ACTION MotorsActualPosition:
// Get Motors Actual Position
rMotorsActualPosition[1] := GVL_Motion.aMotors[1].GetPosition();
rMotorsActualPosition[2] := GVL_Motion.aMotors[2].GetPosition();
rMotorsActualPosition[3] := GVL_Motion.aMotors[3].GetPosition();
rValvesActualPosition[1] := GVL_Motion.aValvesObj[1].GetPosition();
rValvesActualPosition[2] := GVL_Motion.aValvesObj[2].GetPosition();
rValvesActualPosition[3] := GVL_Motion.aValvesObj[3].GetPosition();
rValvesActualPosition[4] := GVL_Motion.aValvesObj[4].GetPosition();
rValvesActualPosition[5] := GVL_Motion.aValvesObj[5].GetPosition();
rPumpsActualPosition[1] := GVL_Motion.aPumpsLinear[1].GetPosition();
rPumpsActualPosition[2] := GVL_Motion.aPumpsLinear[2].GetPosition();
rPumpsActualPosition[3] := GVL_Motion.aPumpsLinear[3].GetPosition();
rPumpsActualPosition[4] := GVL_Motion.aPumpsLinear[4].GetPosition();
rPumpsActualPosition[5] := GVL_Motion.aPumpsLinear[5].GetPosition();
rPumpsActualPosition[6] := GVL_Motion.aPumpsLinear[6].GetPosition();
rPumpsActualPosition[7] := GVL_Motion.aPumpsLinear[7].GetPosition();
rPumpsActualPosition[8] := GVL_Motion.aPumpsLinear[8].GetPosition();
rPumpsActualPosition[9] := GVL_Motion.aPumpsLinear[9].GetPosition();
rPumpsActualPosition[10] := GVL_Motion.aPumpsLinear[10].GetPosition();

//Linear Motors - M1, M2, M3
GVL_Motion.M1Motor.rActualPosition := F_ROUND_REAL(rInput := TO_REAL(rMotorsActualPosition[1]), iDecimalPlaces := 2)* -1;
GVL_Motion.M2Motor.rActualPosition := F_ROUND_REAL(rInput := TO_REAL(rMotorsActualPosition[2]), iDecimalPlaces := 2)* -1;
GVL_Motion.M3Motor.rActualPosition := F_ROUND_REAL(rInput := TO_REAL(rMotorsActualPosition[3]), iDecimalPlaces := 2)* -1;

//Vici Valves - M4 to M8
GVL_Motion.aValves[1].rActualPosition := F_ROUND_REAL(rInput := TO_REAL(rValvesActualPosition[1]), iDecimalPlaces := 2);
GVL_Motion.aValves[2].rActualPosition := F_ROUND_REAL(rInput := TO_REAL(rValvesActualPosition[2]), iDecimalPlaces := 2);
GVL_Motion.aValves[3].rActualPosition := F_ROUND_REAL(rInput := TO_REAL(rValvesActualPosition[3]), iDecimalPlaces := 2);
GVL_Motion.aValves[4].rActualPosition := F_ROUND_REAL(rInput := TO_REAL(rValvesActualPosition[4]), iDecimalPlaces := 2);
GVL_Motion.aValves[5].rActualPosition := F_ROUND_REAL(rInput := TO_REAL(rValvesActualPosition[5]), iDecimalPlaces := 2);

//Linear pumps - 1 to 10
GVL_Motion.aPumps[1].Linear.rActualPosition  := F_ROUND_REAL(rInput := TO_REAL(rPumpsActualPosition[1]), iDecimalPlaces := 2)* -1;
GVL_Motion.aPumps[2].Linear.rActualPosition  := F_ROUND_REAL(rInput := TO_REAL(rPumpsActualPosition[2]), iDecimalPlaces := 2)* -1;
GVL_Motion.aPumps[3].Linear.rActualPosition  := F_ROUND_REAL(rInput := TO_REAL(rPumpsActualPosition[3]), iDecimalPlaces := 2)* -1;
GVL_Motion.aPumps[4].Linear.rActualPosition  := F_ROUND_REAL(rInput := TO_REAL(rPumpsActualPosition[4]), iDecimalPlaces := 2)* -1;
GVL_Motion.aPumps[5].Linear.rActualPosition  := F_ROUND_REAL(rInput := TO_REAL(rPumpsActualPosition[5]), iDecimalPlaces := 2)* -1;
GVL_Motion.aPumps[6].Linear.rActualPosition  := F_ROUND_REAL(rInput := TO_REAL(rPumpsActualPosition[6]), iDecimalPlaces := 2)* -1;
GVL_Motion.aPumps[7].Linear.rActualPosition  := F_ROUND_REAL(rInput := TO_REAL(rPumpsActualPosition[7]), iDecimalPlaces := 2)* -1;
GVL_Motion.aPumps[8].Linear.rActualPosition  := F_ROUND_REAL(rInput := TO_REAL(rPumpsActualPosition[8]), iDecimalPlaces := 2)* -1;
GVL_Motion.aPumps[9].Linear.rActualPosition  := F_ROUND_REAL(rInput := TO_REAL(rPumpsActualPosition[9]), iDecimalPlaces := 2)* -1;
GVL_Motion.aPumps[10].Linear.rActualPosition := F_ROUND_REAL(rInput := TO_REAL(rPumpsActualPosition[10]), iDecimalPlaces := 2)* -1;
END_ACTION

ACTION MotorsJog:
//Manual Motors Moviment

//Manual Moviment motor 1 - Stage Collection Vertical Axis
GVL_Motion.aMotors[1].Jog(bFwd := GVL_HMI.ManualMov.bMotorsJogFwd[1], bBwd := GVL_HMI.ManualMov.bMotorsJogBwd[1]);
//Manual Moviment motor 2 - Sample Recovery Vertical Axis
GVL_Motion.aMotors[2].Jog(bFwd := GVL_HMI.ManualMov.bMotorsJogFwd[2], bBwd := GVL_HMI.ManualMov.bMotorsJogBwd[2]);
//Manual Moviment motor 3 - Sample Recovery Horizontal Axis
GVL_Motion.aMotors[3].Jog(bFwd := GVL_HMI.ManualMov.bMotorsJogFwd[3], bBwd := GVL_HMI.ManualMov.bMotorsJogBwd[3]);

//Manual Moviment M4 - Valve 1 
GVL_Motion.aValvesObj[1].Jog(bFwd := GVL_HMI.ManualMov.bValvesJogFwd[1], bBwd := GVL_HMI.ManualMov.bValvesJogBwd[1]);
//Manual Moviment M5 - Valve 2 
GVL_Motion.aValvesObj[2].Jog(bFwd := GVL_HMI.ManualMov.bValvesJogFwd[2], bBwd := GVL_HMI.ManualMov.bValvesJogBwd[2]);
//Manual Moviment M6 - Valve 3
GVL_Motion.aValvesObj[3].Jog(bFwd := GVL_HMI.ManualMov.bValvesJogFwd[3], bBwd := GVL_HMI.ManualMov.bValvesJogBwd[3]);
//Manual Moviment M7 - Valve 4
GVL_Motion.aValvesObj[4].Jog(bFwd := GVL_HMI.ManualMov.bValvesJogFwd[4], bBwd := GVL_HMI.ManualMov.bValvesJogBwd[4]);
//Manual Moviment M8 - Valve 5
GVL_Motion.aValvesObj[5].Jog(bFwd := GVL_HMI.ManualMov.bValvesJogFwd[5], bBwd := GVL_HMI.ManualMov.bValvesJogBwd[5]);

//Manual Moviment Pump 1 - Linear
GVL_Motion.aPumpsLinear[1].Jog(bFwd := GVL_HMI.ManualMov.bPumpsLinearJogFwd[1], bBwd := GVL_HMI.ManualMov.bPumpsLinearJogBwd[1]);
//Manual Moviment Pump 2 - Linear
GVL_Motion.aPumpsLinear[2].Jog(bFwd := GVL_HMI.ManualMov.bPumpsLinearJogFwd[2], bBwd := GVL_HMI.ManualMov.bPumpsLinearJogBwd[2]);
//Manual Moviment Pump 3 - Linear
GVL_Motion.aPumpsLinear[3].Jog(bFwd := GVL_HMI.ManualMov.bPumpsLinearJogFwd[3], bBwd := GVL_HMI.ManualMov.bPumpsLinearJogBwd[3]);
//Manual Moviment Pump 4 - Linear
GVL_Motion.aPumpsLinear[4].Jog(bFwd := GVL_HMI.ManualMov.bPumpsLinearJogFwd[4], bBwd := GVL_HMI.ManualMov.bPumpsLinearJogBwd[4]);
//Manual Moviment Pump 5 - Linear
GVL_Motion.aPumpsLinear[5].Jog(bFwd := GVL_HMI.ManualMov.bPumpsLinearJogFwd[5], bBwd := GVL_HMI.ManualMov.bPumpsLinearJogBwd[5]);
//Manual Moviment Pump 6 - Linear
GVL_Motion.aPumpsLinear[6].Jog(bFwd := GVL_HMI.ManualMov.bPumpsLinearJogFwd[6], bBwd := GVL_HMI.ManualMov.bPumpsLinearJogBwd[6]);
//Manual Moviment Pump 7 - Linear
GVL_Motion.aPumpsLinear[7].Jog(bFwd := GVL_HMI.ManualMov.bPumpsLinearJogFwd[7], bBwd := GVL_HMI.ManualMov.bPumpsLinearJogBwd[7]);
//Manual Moviment Pump 8 - Linear
GVL_Motion.aPumpsLinear[8].Jog(bFwd := GVL_HMI.ManualMov.bPumpsLinearJogFwd[8], bBwd := GVL_HMI.ManualMov.bPumpsLinearJogBwd[8]);
//Manual Moviment Pump 9 - Linear
GVL_Motion.aPumpsLinear[9].Jog(bFwd := GVL_HMI.ManualMov.bPumpsLinearJogFwd[9], bBwd := GVL_HMI.ManualMov.bPumpsLinearJogBwd[9]);
//Manual Moviment Pump 10 - Linear
GVL_Motion.aPumpsLinear[10].Jog(bFwd := GVL_HMI.ManualMov.bPumpsLinearJogFwd[10], bBwd := GVL_HMI.ManualMov.bPumpsLinearJogBwd[10]);
END_ACTION

METHOD Reset : BOOL
VAR_INPUT
END_VAR
VAR
	i : INT;
END_VAR
// ============================================================================
// PRG_ManualControl.Reset()
// ---------------------------------------------------------------------------
// Clears all manual commands, internal latches and FB states so that
// no manual movement can "resume" automatically when re-entering Manual Mode.
//
// This is a LOGIC reset only:
//  - Does NOT stop axes
//  - Does NOT reset axes
//  - Does NOT enable/disable drives
//
// Intended to be called from SystemInit.
// ============================================================================

// Default return
Reset := FALSE;

// ---------------------------------------------------------------------------
// 1) Reset HMI Manual Motor Commands (M1..M3)
// ---------------------------------------------------------------------------
FOR i := 1 TO 3 DO
    GVL_HMI.aManualMotorsCmd[i].bRun      := FALSE;
    GVL_HMI.aManualMotorsCmd[i].bStop     := FALSE;
    GVL_HMI.aManualMotorsCmd[i].iPosition := 0;
END_FOR

// ---------------------------------------------------------------------------
// 2) Reset HMI Manual Valve Commands (V1..V5)
// ---------------------------------------------------------------------------
FOR i := 1 TO 5 DO
    GVL_HMI.aManualValvesCmd[i].bMove      := FALSE;
    GVL_HMI.aManualValvesCmd[i].bStop      := FALSE;
    GVL_HMI.aManualValvesCmd[i].iTargetPos := 0;
END_FOR

// ---------------------------------------------------------------------------
// 3) Reset HMI Manual Pump Commands (P1..P10)
// ---------------------------------------------------------------------------
FOR i := 1 TO 10 DO
    GVL_HMI.aManualPumpsCmd[i].bActive    := FALSE;
    GVL_HMI.aManualPumpsCmd[i].rSpeed     := 0.0;
    GVL_HMI.aManualPumpsCmd[i].rVolume    := 0.0;
    GVL_HMI.aManualPumpsCmd[i].iDistance  := 0;
END_FOR

GVL_HMI.bRunPumpsBySpeedBt    := FALSE;
GVL_HMI.bRunPumpsByVolumeBt   := FALSE;
GVL_HMI.bRunPumpsByDistanceBt := FALSE;
GVL_HMI.bStopPumpsBt          := FALSE;

// ---------------------------------------------------------------------------
// 4) Reset internal pump control flags and arrays
// ---------------------------------------------------------------------------
bRunPumpsBySpeed    := FALSE;
bRunPumpsByVolume   := FALSE;
bRunPumpsByDistance := FALSE;

FOR i := 1 TO 10 DO
    aPumpsActivated[i] := FALSE;
    aPumpsSpeed[i]     := 0.0;
    aPumpsVolume[i]    := 0.0;
    aPumpsDistance[i]  := 0;
END_FOR

// ---------------------------------------------------------------------------
// 5) Reset interlock and auxiliary variables
// ---------------------------------------------------------------------------
bAllowMoveM2 := TRUE;
iTargetPosM2 := 0;
iM3Position  := 0;
rActualPosM3 := 0.0;

// ---------------------------------------------------------------------------
// 6) Reset FBs with internal state
// ---------------------------------------------------------------------------
fbPumpsController.Reset();   // assumes your FB has a Reset() method

// ---------------------------------------------------------------------------
// 7) Finalize
// ---------------------------------------------------------------------------
Reset := TRUE;
END_METHOD

END_PROGRAM

// ---- POUs/Functions/F_ROUND_REAL.TcPOU
FUNCTION F_ROUND_REAL : LREAL
VAR_INPUT
	rInput : LREAL;
  	iDecimalPlaces : INT;
END_VAR
VAR
	rFactor : LREAL;
    rScaled : LREAL;
    rRounded : LREAL;
END_VAR

rFactor := EXPT(10.0, iDecimalPlaces);         // Ex: 100.0 for 2 digits
rScaled := rInput * rFactor;

IF rScaled >= 0.0 THEN
    rRounded := TRUNC(rScaled + 0.5);
ELSE
    rRounded := TRUNC(rScaled - 0.5);
END_IF

F_ROUND_REAL := rRounded / rFactor;

END_FUNCTION

// ---- POUs/1. MachineControl/PRG_StoppedState.TcPOU
PROGRAM PRG_StoppedState

VAR_OUTPUT
    bStopAllMotorsDone : BOOL := FALSE; // TRUE when ALL axes (motors, valves, rotary pumps,
                     					// linear pumps) have completely finished stopping.
	                      				// Used by PRG_MasterControl to release SystemInit.
END_VAR

VAR
    // ------------------------------------------------------------------------
    // 1) HMI / Visual Feedback
    // ------------------------------------------------------------------------
    fbBlinkStartButton : FB_Blink;  // Blink logic for the Start button indicator
    
    // ------------------------------------------------------------------------
    // 2) Master Stop Execution Control
    // ------------------------------------------------------------------------
    bStopAllMotorsRequest : BOOL := FALSE;  
    // One-shot latch:
    // FALSE → stop request not yet triggered
    // TRUE  → stop request already armed; stop routine executing

    // ------------------------------------------------------------------------
    // 3) Per-axis STOP flags
    //    These arrays are used by ACTION ACT_StopAllMotors.
    //    TRUE  → axis still must be stopped (Stop() still being executed)
    //    FALSE → axis already fully stopped
    // ------------------------------------------------------------------------
    bStopMotors        : ARRAY[1..3]  OF BOOL;   // Linear motors M1..M3
    bStopValves        : ARRAY[1..5]  OF BOOL;   // Valves V1..V5
    bStopLinearPumps   : ARRAY[1..10] OF BOOL;   // Linear pump axes
    bStopRotaryPumps   : ARRAY[1..10] OF BOOL;   // Rotary pump axes

    // ------------------------------------------------------------------------
    // 4) Axis Status Structures
    //    Captured during ACTION ACT_ResetErrorMotors.
    // ------------------------------------------------------------------------
    stMotorStatus       : ARRAY[1..3]  OF ST_AxisReadStatus;
    stValveStatus       : ARRAY[1..5]  OF ST_AxisReadStatus;
    stLinearPumpStatus  : ARRAY[1..10] OF ST_AxisReadStatus;
    stRotaryPumpStatus  : ARRAY[1..10] OF ST_AxisReadStatus;

    // ------------------------------------------------------------------------
    // 5) Reset request guards for each axis
    //    TRUE  → Reset already attempted
    //    FALSE → Reset() still allowed to be triggered once
    // ------------------------------------------------------------------------
    aResetMotors       : ARRAY[1..3]  OF BOOL;
    aResetValves       : ARRAY[1..5]  OF BOOL;
    aResetLinearPumps  : ARRAY[1..10] OF BOOL;
    aResetRotaryPumps  : ARRAY[1..10] OF BOOL;

    // ------------------------------------------------------------------------
    // 6) Stop Monitoring Flags (used inside the refactored ACT_StopAllMotors)
    // ------------------------------------------------------------------------
    iAxis                    : INT;   // Generic loop index
    bIsNotMoving             : BOOL;  // Temporary axis movement flag
    bAllMotorsStopped        : BOOL;  // Group completion flags
    bAllValvesStopped        : BOOL;
    bAllRotaryPumpsStopped   : BOOL;
    bAllLinearPumpsStopped   : BOOL;

    // ------------------------------------------------------------------------
    // 7) Global Reset / StateMachine Control Flags
    // ------------------------------------------------------------------------ 
    bAllMotorsStop    : BOOL := FALSE;  // TRUE when all axes reached iNotMoving
    bAutoCycleReset   : BOOL := FALSE;  // TRUE when PRG_StateMachine.Reset() finished
    bCalibrationReset : BOOL := FALSE;  // TRUE when PRG_Calibration.Reset() finished
    bAllResetsDone    : BOOL := FALSE;  // TRUE when everything above is completed
	
	bAStopLogicLatchesDone	: BOOL := FALSE; // TRUE when as latches and flags were set to false
	
	i : INT; 

END_VAR

// ============================================================================
// PRG_StoppedState
// ----------------------------------------------------------------------------
// This program is executed while the machine is in the "Stopped" state.
// Responsibilities:
//  - Make the Start button blink when it is safe to start again
//  - Stop all axes (motors, valves, pumps) in a controlled way
//  - Reset axis errors
//  - Reset the AutoCycle and Calibration state machines
//  - Inform MasterControl when everything is fully reset (bAllResetsDone)
// ============================================================================

// ---------------------------------------------------------------------------
// Start Button Blink
//  - Blink only when: Safety is OK, all axes are stopped, and all resets done
//  - Output: GVL_IO.gDigOutputs.bStartIndicator
// ---------------------------------------------------------------------------
IF GVL_Safety.bSafetyEnable AND bStopAllMotorsDone AND bAStopLogicLatchesDone (*AND bAllResetsDone AND bCalibrationReset*) THEN 
    fbBlinkStartButton( bEnable := TRUE, tPeriod := T#1S );
ELSE
    fbBlinkStartButton( bEnable := FALSE, tPeriod := T#1S );
END_IF

GVL_IO.gDigOutputs.bStartIndicator := fbBlinkStartButton.bBlink;

// ---------------------------------------------------------------------------
// Reset axis errors
//  - Only executed after ALL motors have been confirmed as stopped
//  - This avoids resetting drives while they are still trying to stop
// ---------------------------------------------------------------------------
(*IF bAllMotorsStop THEN
    ACT_ResetErrorMotors();
END_IF
*)

IF NOT bAStopLogicLatchesDone THEN ACT_ResetCommandFlags(); END_IF


// ---------------------------------------------------------------------------
// Stop all axes
//  - This action:
//      * Sets stop requests for every axis (one-shot)
//      * Calls Stop() for each axis while it is moving
//      * Monitors when all stop requests are cleared
//      * Sets bStopAllMotorsDone when everything is stopped
// ---------------------------------------------------------------------------
ACT_StopAllMotors();

IF bStopAllMotorsDone THEN
    bAllMotorsStop := TRUE;     // All axes are now in a "not moving" state
END_IF
(*
// ---------------------------------------------------------------------------
// Reset AutoCycle State Machine
//  - PRG_StateMachine.Reset() should internally clear its own flags and states
//  - This is called until it returns TRUE once
// ---------------------------------------------------------------------------
IF NOT bAutoCycleReset THEN
    bAutoCycleReset := PRG_AutoCycle.Reset();
END_IF

// ---------------------------------------------------------------------------
// Reset Calibration Program
//  - PRG_Calibration.Reset() behaves similarly to PRG_StateMachine.Reset()
// ---------------------------------------------------------------------------
IF NOT bCalibrationReset THEN
    bCalibrationReset := PRG_Calibration.Reset();
END_IF

// ---------------------------------------------------------------------------
// Global done flag
//  - Used by MasterControl to know when StoppedState finished its job
//  - Only TRUE when:
//      * All axes are stopped   (bStopAllMotorsDone)
//      * AutoCycle reset is ok  (bAutoCycleReset)
//      * Calibration reset is ok(bCalibrationReset)
// ---------------------------------------------------------------------------
bAllResetsDone := bStopAllMotorsDone AND bAutoCycleReset AND bCalibrationReset;
*)

(* Before Tidy up from 05/12 
//Start Button Blink ------------------------------------------------
IF GVL_Safety.bSafetyEnable AND bStopAllMotorsDone AND bAllResetsDone THEN 
	fbBlinkStartButton( bEnable := TRUE, tPeriod := T#1S );
ELSE
	fbBlinkStartButton( bEnable := FALSE, tPeriod := T#1S );
END_IF

GVL_IO.gDigOutputs.bStartIndicator := fbBlinkStartButton.bBlink;

//Action to check if is there any motors with erros and reset them  
IF bAllMotorsStop THEN
	ACT_ResetErrorMotors();
END_IF

//Action to stop all motors 
ACT_StopAllMotors();

IF bStopAllMotorsDone THEN
	bAllMotorsStop := TRUE;
END_IF

//State Machine Reset
IF NOT bAutoCycleReset THEN
	bAutoCycleReset := PRG_StateMachine.Reset();
END_IF

//Calibration PRG Reset
IF NOT bCalibrationReset THEN
	bCalibrationReset := PRG_Calibration.Reset();
END_IF

bAllResetsDone := bStopAllMotorsDone AND bAutoCycleReset AND bCalibrationReset; *)

ACTION ACT_ResetCommandFlags:
(*
    Action: ACT_ResetCommandFlags
    Purpose:
        Clear all HMI command flags and internal latched commands that might remain TRUE
        after an abnormal interruption (STOP/Abort), preventing unintended auto-start
        when re-entering a mode.

    Where to call:
        - PRG_StoppedState (first scan / when entering STOPPED)
        - PRG_SystemInit (first scan / at init start)

    Notes:
        - This action is safe to call repeatedly (idempotent).
        - Adjust array bounds if your project differs.
*)

// ============================================================
// 1) Calibration - HMI triggers (buttons / commands)
// ============================================================
GVL_HMI.bStartCalibrationBt        := FALSE;

GVL_HMI.bCalLeakTestButton         := FALSE;
GVL_HMI.bCalPressureUpSystemBt     := FALSE;
GVL_HMI.bCalHoldSysPressureBt      := FALSE;
GVL_HMI.bCalStopLeakTestBt         := FALSE;

GVL_HMI.bCalLinearPumpsEnableBt    := FALSE;
GVL_HMI.bCalLinearPumpsHomeBt      := FALSE;
GVL_HMI.bCalLinearPumpsMoveBt      := FALSE;
GVL_HMI.bCalLinearPumpsStopBt      := FALSE;
GVL_HMI.bCalLinearPumpsDirty       := FALSE;

GVL_HMI.bCalMoveValves             := FALSE;
GVL_HMI.bCalMoveM1Motor            := FALSE;

// Scale / CalBox popups / acknowledge flags
GVL_HMI.bScaleNeedsAtention        := FALSE;
GVL_HMI.bScaleFixed                := FALSE;
GVL_HMI.bCalBoxNeedsAttention      := FALSE;
GVL_HMI.bCalBoxFixed               := FALSE;


// ============================================================
// 2) Calibration - internal latches (must be cleared on STOP/Init)
// ============================================================
GVL_Calibration.bStartCalibration      := FALSE;
GVL_Calibration.bAbortCalibration      := FALSE;
GVL_Calibration.bStartCreationCalJson  := FALSE;


// ============================================================
// 3) Manual Mode - motors / valves / pumps command arrays
// ============================================================

// Manual motors (adjust bounds if needed)
FOR i := 1 TO 3 DO
    GVL_HMI.aManualMotorsCmd[i].bRun  := FALSE;
    GVL_HMI.aManualMotorsCmd[i].bStop := FALSE;
END_FOR

// Manual valves
FOR i := 1 TO 5 DO
    GVL_HMI.aManualValvesCmd[i].bMove := FALSE;
    GVL_HMI.aManualValvesCmd[i].bStop := FALSE;
END_FOR

// Global pump buttons
GVL_HMI.bRunPumpsBySpeedBt  := FALSE;
GVL_HMI.bRunPumpsByVolumeBt := FALSE;

// Per-pump commands
FOR i := 1 TO 10 DO
    GVL_HMI.aManualPumpsCmd[i].bRunBySpeed  := FALSE;
    GVL_HMI.aManualPumpsCmd[i].bRunByVolume := FALSE;
    GVL_HMI.aManualPumpsCmd[i].bStop        := FALSE;
    GVL_HMI.aManualPumpsCmd[i].bActive      := FALSE;
END_FOR


// ============================================================
// 4) AutoCycle - popup/start/hold commands
// ============================================================
GVL_HMI.bShowAutoCyclePopup     	:= FALSE;
GVL_HMI.bStartAutoCycleButton   	:= FALSE;
GVL_HMI.bSystemReady_ReqAutoCycle 	:= FALSE;

GVL_HMI.bAutoCycleHoldReq       	:= FALSE;
GVL_HMI.bAutoCycleHoldActive    	:= FALSE;
GVL_HMI.bAutoCycleHoldPopup     	:= FALSE;
GVL_HMI.bAutoCycleContinueCmd   	:= FALSE;
GVL_HMI.bAutoCycleCancelCmd     	:= FALSE;


// ============================================================
// 5) Finishing
// ============================================================
bAStopLogicLatchesDone := TRUE;
END_ACTION

ACTION ACT_ResetErrorMotors:
// ============================================================================
// ACT_ResetErrorMotors
// ----------------------------------------------------------------------------
// Purpose:
//  1) Read status from all axis wrappers (motors, valves, pumps)
//  2) For each axis that is in Error, call its Reset() method once
//     - The aReset* arrays guarantee we do not repeatedly call Reset()
//     - Reset() is expected to return TRUE when the reset command has been sent
// ============================================================================

// ---------------------------------------------------------------------------
// 1) Read status from all axis wrappers
// ---------------------------------------------------------------------------

// Linear motors (M1..M3)
FOR iAxis := 1 TO 3 DO
    stMotorStatus[iAxis] := GVL_Motion.aMotors[iAxis].ReadStatus();
END_FOR

// Valves servo motors (V1..V5)
FOR iAxis := 1 TO 5 DO
    stValveStatus[iAxis] := GVL_Motion.aValvesObj[iAxis].ReadStatus();
END_FOR

// Linear pump motors (1..10)
FOR iAxis := 1 TO 10 DO
    stLinearPumpStatus[iAxis] := GVL_Motion.aPumpsLinear[iAxis].ReadStatus();
END_FOR

// Rotary pump motors (1..10)
FOR iAxis := 1 TO 10 DO
    stRotaryPumpStatus[iAxis] := GVL_Motion.aPumpsRotary[iAxis].ReadStatus();
END_FOR

// ---------------------------------------------------------------------------
// 2) For each axis in Error = TRUE, call Reset() once
//    The flag arrays (aReset*) are used as "one-shot" guards per axis.
// ---------------------------------------------------------------------------

// Linear motors

IF stMotorStatus[1].Error OR GVL_Motion.M1Motor.bMotionCommandsLocked THEN
	IF NOT aResetMotors[1] THEN
		aResetMotors[1] := GVL_Motion.aMotors[1].Reset();
	END_IF
END_IF

IF stMotorStatus[2].Error OR GVL_Motion.M2Motor.bMotionCommandsLocked THEN
	IF NOT aResetMotors[2] THEN
		aResetMotors[2] := GVL_Motion.aMotors[2].Reset();
	END_IF
END_IF

IF stMotorStatus[3].Error OR GVL_Motion.M3Motor.bMotionCommandsLocked THEN
	IF NOT aResetMotors[3] THEN
		aResetMotors[3] := GVL_Motion.aMotors[3].Reset();
	END_IF
END_IF

// Valves servo motors
FOR iAxis := 1 TO 5 DO
    IF stValveStatus[iAxis].Error OR GVL_Motion.aValves[iAxis].bMotionCommandsLocked THEN
        IF NOT aResetValves[iAxis] THEN
            aResetValves[iAxis] := GVL_Motion.aValvesObj[iAxis].Reset();
        END_IF
    END_IF
END_FOR

// Linear pump motors
FOR iAxis := 1 TO 10 DO
    IF stLinearPumpStatus[iAxis].Error OR GVL_Motion.aPumps[iAxis].Linear.bMotionCommandsLocked THEN
        IF NOT aResetLinearPumps[iAxis] THEN
            aResetLinearPumps[iAxis] := GVL_Motion.aPumpsLinear[iAxis].Reset();
        END_IF
    END_IF
END_FOR

// Rotary pump motors
FOR iAxis := 1 TO 10 DO
    IF stRotaryPumpStatus[iAxis].Error OR GVL_Motion.aPumps[iAxis].Rotary.bMotionCommandsLocked THEN
        IF NOT aResetRotaryPumps[iAxis] THEN
            aResetRotaryPumps[iAxis] := GVL_Motion.aPumpsRotary[iAxis].Reset();
        END_IF
    END_IF
END_FOR


(* Before Tidy up from 05/12
//Getting status from all motors
//Linear Motors
FOR i := 1 TO 3 DO
	stMotorStatus[i] := GVL_Motion.aMotors[i].ReadStatus();
END_FOR
//Valves Servo Motors
FOR i := 1 TO 5 DO
	stValveStatus[i] := GVL_Motion.aValvesObj[i].ReadStatus();
END_FOR
//Linear Pumps Motors
FOR i := 1 TO 10 DO
	stLinearPumpStatus[i] := GVL_Motion.aPumpsLinear[i].ReadStatus();
END_FOR
//Rotary Pumps Motors
FOR i := 1 TO 10 DO
	stRotaryPumpStatus[i] := GVL_Motion.aPumpsRotary[i].ReadStatus();
END_FOR

//Reset the motors that are in error
//Linear Motors
FOR i := 1 TO 3 DO
	IF stMotorStatus[i].Error THEN
		IF NOT aResetMotors[i] THEN
			aResetMotors[i] := GVL_Motion.aMotors[i].Reset();
		END_IF
	END_IF
END_FOR
//Valves Servo Motors
FOR i := 1 TO 5 DO
	IF stValveStatus[i].Error THEN
		IF NOT aResetValves[i] THEN
			aResetValves[i] := GVL_Motion.aValvesObj[i].Reset();
		END_IF
	END_IF
END_FOR
//Linear Pumps Motors
FOR i := 1 TO 10 DO
	IF stLinearPumpStatus[i].Error THEN
		IF NOT aResetLinearPumps[i] THEN
			aResetLinearPumps[i] := GVL_Motion.aPumpsLinear[i].Reset();
		END_IF
	END_IF
END_FOR
//Rotary Pumps Motors
FOR i := 1 TO 10 DO
	IF stRotaryPumpStatus[i].Error THEN
		IF NOT aResetRotaryPumps[i] THEN
			aResetRotaryPumps[i] := GVL_Motion.aPumpsRotary[i].Reset();
		END_IF
	END_IF
END_FOR*)
END_ACTION

ACTION ACT_StopAllMotors:
// ============================================================================
// ACT_StopAllMotors (Refactored)
// ----------------------------------------------------------------------------
// Purpose:
//  - Trigger a controlled stop for all motion axes:
//      * Linear motors (M1..M3)
//      * Valves servo motors (V1..V5)
//      * Rotary pumps (1..10)
//      * Linear pumps (1..10)
//  - Stop logic:
//      1) On first call (bStopAllMotorsRequest = FALSE), set all stop flags = TRUE
//      2) For each axis that is still moving, call its Stop() method
//      3) When Stop() returns TRUE, clear the corresponding flag to FALSE
//      4) When all flags are FALSE, set bStopAllMotorsDone = TRUE
// ============================================================================


// ---------------------------------------------------------------------------
// 1) One-shot: arm stop request for all axes
//    This block runs only once per StoppedState sequence.
// ---------------------------------------------------------------------------
IF NOT bStopAllMotorsRequest THEN
    // Linear motors
    bStopMotors[1] := NOT GVL_Motion.M1Motor.iNotMoving;      // Stop request for each linear motor
	bStopMotors[2] := NOT GVL_Motion.M2Motor.iNotMoving; 
	bStopMotors[3] := NOT GVL_Motion.M3Motor.iNotMoving; 
	
    // Valves servo motors
    FOR iAxis := 1 TO 5 DO
        bStopValves[iAxis] := NOT GVL_Motion.aValves[iAxis].iNotMoving;      // Stop request for each valve axis
    END_FOR

    // Linear pumps
    FOR iAxis := 1 TO 10 DO
        bStopLinearPumps[iAxis] := NOT GVL_Motion.aPumps[iAxis].Linear.iNotMoving; // Stop request for each linear pump axis
    END_FOR

    // Rotary pumps
    FOR iAxis := 1 TO 10 DO
        bStopRotaryPumps[iAxis] := NOT GVL_Motion.aPumps[iAxis].Rotary.iNotMoving; // Stop request for each rotary pump axis
    END_FOR
    
    bStopAllMotorsRequest := TRUE;       // One-shot armed
    bStopAllMotorsDone    := FALSE;      // Not done yet
END_IF


// ---------------------------------------------------------------------------
// 2) Call Stop() for each axis while it is still moving
//    Strategy:
//      - If axis is moving (iNotMoving = FALSE), keep requesting Stop()
//      - When Stop() returns TRUE, we clear the stop flag to FALSE
//      - If axis is already not moving, force the flag to FALSE
// ---------------------------------------------------------------------------

// --- Linear motors Stop - M1 to M3 -----------------------------------------
IF bStopMotors[1] THEN
	IF NOT GVL_Motion.M1Motor.iNotMoving THEN
		bStopMotors[1] := NOT GVL_Motion.aMotors[1].Stop();
	ELSE
		bStopMotors[1] := FALSE;
	END_IF
END_IF

IF bStopMotors[2] THEN
	IF NOT GVL_Motion.M2Motor.iNotMoving THEN
		bStopMotors[2] := NOT GVL_Motion.aMotors[2].Stop();
	ELSE
		bStopMotors[2] := FALSE;
	END_IF
END_IF
	

IF bStopMotors[3] THEN
	IF NOT GVL_Motion.M3Motor.iNotMoving THEN
		bStopMotors[3] := NOT GVL_Motion.aMotors[3].Stop();
	ELSE
		bStopMotors[3] := FALSE;
	END_IF
END_IF
	
// --- Valves Servo Motors Stop - V1 to V5 -----------------------------------
FOR iAxis := 1 TO 5 DO
	IF bStopValves[iAxis] THEN
		IF NOT GVL_Motion.aValves[iAxis].iNotMoving THEN
			bStopValves[iAxis] := NOT GVL_Motion.aValvesObj[iAxis].Stop();
		ELSE
			bStopValves[iAxis] := FALSE;
		END_IF
	END_IF
END_FOR


// --- Rotary Pumps Stop - 1 to 10 -------------------------------------------
//  - aPumps[x].Rotary.iNotMoving: feedback "axis moving" for each rotary pump
//  - aPumpsRotary[x].Stop(): Stop method on the pump rotary axis wrapper
FOR iAxis := 1 TO 10 DO
	IF  bStopRotaryPumps[iAxis] THEN
		IF NOT GVL_Motion.aPumps[iAxis].Rotary.iNotMoving THEN
			bStopRotaryPumps[iAxis] := NOT GVL_Motion.aPumpsRotary[iAxis].Stop();
		ELSE
			bStopRotaryPumps[iAxis] := FALSE;
		END_IF
	END_IF
END_FOR


// --- Linear Pumps Stop - 1 to 10 -------------------------------------------
//  - aPumps[x].Linear.iNotMoving: feedback "axis moving" for each linear pump
//  - aPumpsLinear[x].Stop(): Stop method on the linear pump axis wrapper
FOR iAxis := 1 TO 10 DO
	IF bStopLinearPumps[iAxis] THEN
		IF NOT GVL_Motion.aPumps[iAxis].Linear.iNotMoving THEN
			bStopLinearPumps[iAxis] := NOT GVL_Motion.aPumpsLinear[iAxis].Stop();
		ELSE
			bStopLinearPumps[iAxis] := FALSE;
		END_IF
	END_IF
END_FOR


// ---------------------------------------------------------------------------
// 3) Global "done" condition for stopping all axes
//    When no stop flag is active in any group, all axes are considered stopped.
// ---------------------------------------------------------------------------

// Check linear motors

bAllMotorsStopped := NOT bStopMotors[1] AND NOT bStopMotors[2] AND NOT bStopMotors[3];


// Check valves
bAllValvesStopped := TRUE;
FOR iAxis := 1 TO 5 DO
    bAllValvesStopped := bAllValvesStopped AND NOT bStopValves[iAxis];
END_FOR

// Check rotary pumps
bAllRotaryPumpsStopped := TRUE;
FOR iAxis := 1 TO 10 DO
    bAllRotaryPumpsStopped := bAllRotaryPumpsStopped AND NOT bStopRotaryPumps[iAxis];
END_FOR

// Check linear pumps
bAllLinearPumpsStopped := TRUE;
FOR iAxis := 1 TO 10 DO
    bAllLinearPumpsStopped := bAllLinearPumpsStopped AND NOT bStopLinearPumps[iAxis];
END_FOR

// Final global flag
bStopAllMotorsDone := bAllMotorsStopped
                      AND bAllValvesStopped
                      AND bAllRotaryPumpsStopped
                      AND bAllLinearPumpsStopped;


(* Before Tidy up from 05/12
//Stop all motors. Linear, valves, pumps.
IF NOT bStopAllMotorsRequest THEN
	FOR i := 1 TO 3 DO
		bStopMotors[i] := TRUE; //Stop Request for every motor turn true
	END_FOR
	FOR i := 1 TO 5 DO
		bStopValves[i] := TRUE;
	END_FOR
	FOR i := 1 TO 10 DO
		bStopLinearPumps[i] := TRUE;
	END_FOR
	FOR i := 1 TO 10 DO
		bStopRotaryPumps[i] := TRUE;
	END_FOR
	
	bStopAllMotorsRequest	:= TRUE;
	bStopAllMotorsDone		:= FALSE;
END_IF

//Every Motor Method Stop() call
//Linear Motors Stop - M1 to M3
IF NOT GVL_Motion.M1Motor.iNotMoving THEN
	bStopMotors[1] := NOT GVL_Motion.aMotors[1].Stop();
ELSE
	bStopMotors[1] := FALSE;
END_IF

IF NOT GVL_Motion.M2Motor.iNotMoving THEN
	bStopMotors[2] := NOT GVL_Motion.aMotors[2].Stop();
ELSE
	bStopMotors[2] := FALSE;
END_IF


IF NOT GVL_Motion.M3Motor.iNotMoving THEN
	bStopMotors[3] := NOT GVL_Motion.aMotors[3].Stop();
ELSE
	bStopMotors[3] := FALSE;
END_IF

//Valve Servo Motors Stop - M4 to M8
IF NOT GVL_Motion.aValves[1].iNotMoving THEN
	bStopValves[1] := NOT GVL_Motion.aValvesObj[1].Stop();
ELSE
	bStopValves[1] := FALSE;
END_IF

IF NOT GVL_Motion.aValves[2].iNotMoving THEN
	bStopValves[2] := NOT GVL_Motion.aValvesObj[2].Stop();
ELSE
	bStopValves[2] := FALSE;
END_IF

IF NOT GVL_Motion.aValves[3].iNotMoving THEN
	bStopValves[3] := NOT GVL_Motion.aValvesObj[3].Stop();
ELSE
	bStopValves[3] := FALSE;
END_IF

IF NOT GVL_Motion.aValves[4].iNotMoving THEN
	bStopValves[4] := NOT GVL_Motion.aValvesObj[4].Stop();
ELSE
	bStopValves[4] := FALSE;
END_IF

IF NOT GVL_Motion.aValves[5].iNotMoving THEN
	bStopValves[5] := NOT GVL_Motion.aValvesObj[5].Stop();
ELSE
	bStopValves[5] := FALSE;
END_IF

//Rotary Pumps Stop - 1 to 10
IF NOT GVL_Motion.aPumps[1].Rotary.iNotMoving THEN
	bStopRotaryPumps[1] := NOT GVL_Motion.aPumpsRotary[1].Stop();
ELSE
	bStopRotaryPumps[1] := FALSE;
END_IF

IF NOT GVL_Motion.aPumps[2].Rotary.iNotMoving THEN
	bStopRotaryPumps[2] := NOT GVL_Motion.aPumpsRotary[2].Stop();
ELSE
	bStopRotaryPumps[2] := FALSE;
END_IF

IF NOT GVL_Motion.aPumps[3].Rotary.iNotMoving THEN
	bStopRotaryPumps[3] := NOT GVL_Motion.aPumpsRotary[3].Stop();
ELSE
	bStopRotaryPumps[3] := FALSE;
END_IF

IF NOT GVL_Motion.aPumps[4].Rotary.iNotMoving THEN
	bStopRotaryPumps[4] := NOT GVL_Motion.aPumpsRotary[4].Stop();
ELSE
	bStopRotaryPumps[4] := FALSE;
END_IF

IF NOT GVL_Motion.aPumps[5].Rotary.iNotMoving THEN
	bStopRotaryPumps[5] := NOT GVL_Motion.aPumpsRotary[5].Stop();
ELSE
	bStopRotaryPumps[5] := FALSE;
END_IF

IF NOT GVL_Motion.aPumps[6].Rotary.iNotMoving THEN
	bStopRotaryPumps[6] := NOT GVL_Motion.aPumpsRotary[6].Stop();
ELSE
	bStopRotaryPumps[6] := FALSE;
END_IF

IF NOT GVL_Motion.aPumps[7].Rotary.iNotMoving THEN
	bStopRotaryPumps[7] := NOT GVL_Motion.aPumpsRotary[7].Stop();
ELSE
	bStopRotaryPumps[7] := FALSE;
END_IF

IF NOT GVL_Motion.aPumps[8].Rotary.iNotMoving THEN
	bStopRotaryPumps[8] := NOT GVL_Motion.aPumpsRotary[8].Stop();
ELSE
	bStopRotaryPumps[8] := FALSE;
END_IF

IF NOT GVL_Motion.aPumps[9].Rotary.iNotMoving THEN
	bStopRotaryPumps[9] := NOT GVL_Motion.aPumpsRotary[9].Stop();
ELSE
	bStopRotaryPumps[9] := FALSE;
END_IF

IF NOT GVL_Motion.aPumps[10].Rotary.iNotMoving THEN
	bStopRotaryPumps[10] := NOT GVL_Motion.aPumpsRotary[10].Stop();
ELSE
	bStopRotaryPumps[10] := FALSE;
END_IF

//Linear Pumps Stop - 1 to 10
IF NOT GVL_Motion.aPumps[1].Linear.iNotMoving THEN
	bStopLinearPumps[1] := NOT GVL_Motion.aPumpsLinear[1].Stop();
ELSE
	bStopLinearPumps[1] := FALSE;
END_IF

IF NOT GVL_Motion.aPumps[2].Linear.iNotMoving THEN
	bStopLinearPumps[2] := NOT GVL_Motion.aPumpsLinear[2].Stop();
ELSE
	bStopLinearPumps[2] := FALSE;
END_IF

IF NOT GVL_Motion.aPumps[3].Linear.iNotMoving THEN
	bStopLinearPumps[3] := NOT GVL_Motion.aPumpsLinear[3].Stop();
ELSE
	bStopLinearPumps[3] := FALSE;
END_IF

IF NOT GVL_Motion.aPumps[4].Linear.iNotMoving THEN
	bStopLinearPumps[4] := NOT GVL_Motion.aPumpsLinear[4].Stop();
ELSE
	bStopLinearPumps[4] := FALSE;
END_IF

IF NOT GVL_Motion.aPumps[5].Linear.iNotMoving THEN
	bStopLinearPumps[5] := NOT GVL_Motion.aPumpsLinear[5].Stop();
ELSE
	bStopLinearPumps[5] := FALSE;
END_IF

IF NOT GVL_Motion.aPumps[6].Linear.iNotMoving THEN
	bStopLinearPumps[6] := NOT GVL_Motion.aPumpsLinear[6].Stop();
ELSE
	bStopLinearPumps[6] := FALSE;
END_IF

IF NOT GVL_Motion.aPumps[7].Linear.iNotMoving THEN
	bStopLinearPumps[7] := NOT GVL_Motion.aPumpsLinear[7].Stop();
ELSE
	bStopLinearPumps[7] := FALSE;
END_IF

IF NOT GVL_Motion.aPumps[8].Linear.iNotMoving THEN
	bStopLinearPumps[8] := NOT GVL_Motion.aPumpsLinear[8].Stop();
ELSE
	bStopLinearPumps[8] := FALSE;
END_IF

IF NOT GVL_Motion.aPumps[9].Linear.iNotMoving THEN
	bStopLinearPumps[9] := NOT GVL_Motion.aPumpsLinear[9].Stop();
ELSE
	bStopLinearPumps[9] := FALSE;
END_IF

IF NOT GVL_Motion.aPumps[10].Linear.iNotMoving THEN
	bStopLinearPumps[10] := NOT GVL_Motion.aPumpsLinear[10].Stop();
ELSE
	bStopLinearPumps[10] := FALSE;
END_IF

IF NOT bStopMotors[1] AND NOT bStopMotors[2] AND NOT bStopMotors[3] THEN
	IF NOT bStopValves[1] AND NOT bStopValves[2] AND NOT bStopValves[3] AND NOT bStopValves[4] AND NOT bStopValves[5] THEN
		IF NOT bStopRotaryPumps[1] AND NOT bStopRotaryPumps[2] AND NOT bStopRotaryPumps[3] AND NOT bStopRotaryPumps[4] AND NOT bStopRotaryPumps[5] AND NOT bStopRotaryPumps[6] AND NOT bStopRotaryPumps[7] AND NOT bStopRotaryPumps[8] AND NOT bStopRotaryPumps[9] AND NOT bStopRotaryPumps[10] THEN
			IF NOT bStopLinearPumps[1] AND NOT bStopLinearPumps[2] AND NOT bStopLinearPumps[3] AND NOT bStopLinearPumps[4] AND NOT bStopLinearPumps[5] AND NOT bStopLinearPumps[6] AND NOT bStopLinearPumps[7] AND NOT bStopLinearPumps[8] AND NOT bStopLinearPumps[9] AND NOT bStopLinearPumps[10] THEN
				bStopAllMotorsDone		:= TRUE;
			END_IF
		END_IF
	END_IF
END_IF
*)
END_ACTION

METHOD Reset : BOOL
VAR_INPUT
END_VAR
// ============================================================================
// Reset()
// ----------------------------------------------------------------------------
// Purpose:
//  - Clear all internal flags and arrays of PRG_StoppedState
//  - Prepare this program to run a new full stopped-sequence
// Behavior:
//  - Sets all internal booleans and arrays to FALSE
//  - Returns TRUE once, when the reset conditions are satisfied
//    (here: simply when there is no stop request and no "done" flag)
// ============================================================================

// ---------------------------------------------------------------------------
// 1) Reset main flags
// ---------------------------------------------------------------------------
bStopAllMotorsRequest := FALSE;
bStopAllMotorsDone    := FALSE;

bAllMotorsStop          := FALSE;
bAutoCycleReset         := FALSE;
bCalibrationReset       := FALSE;
bAllResetsDone          := FALSE;
bAStopLogicLatchesDone  := FALSE;

// ---------------------------------------------------------------------------
// 2) Reset arrays used in error reset / stop logic
// ---------------------------------------------------------------------------
// Motors reset flags
FOR iAxis := 1 TO 3 DO
    aResetMotors[iAxis] := FALSE;
END_FOR

// Valves reset flags
FOR iAxis := 1 TO 5 DO
    aResetValves[iAxis] := FALSE;
END_FOR

// Linear pumps reset flags
FOR iAxis := 1 TO 10 DO
    aResetLinearPumps[iAxis] := FALSE;
END_FOR

// Rotary pumps reset flags
FOR iAxis := 1 TO 10 DO
    aResetRotaryPumps[iAxis] := FALSE;
END_FOR

// ---------------------------------------------------------------------------
// 3) Return value
//    - With the current logic, right after executing this method
//      both bStopAllMotorsRequest and bStopAllMotorsDone are FALSE
//      so Reset = TRUE will be returned.
// ---------------------------------------------------------------------------
IF NOT bStopAllMotorsRequest AND NOT bStopAllMotorsDone THEN
    Reset := TRUE;
    RETURN;
ELSE
    Reset := FALSE;
END_IF
END_METHOD

END_PROGRAM

// ---- POUs/1. MachineControl/PRG_SystemReady.TcPOU
PROGRAM PRG_SystemReady
VAR_OUTPUT
	bSystemReadyToStart : BOOL;      // TRUE when machine is ready to accept Start 	 	
END_VAR
VAR
	fbBlinkStartButton      : FB_Blink;
    fbBlinkMachineModeName  : FB_Blink;

    bRecipeCorrectLoaded    : BOOL := FALSE;
    bSettingsCorrectLoaded  : BOOL := FALSE;

    rTrigStartButton        : R_TRIG;    // Rising edge for main Start button
    rTrigPopupStartBtn      : R_TRIG;    // Rising edge for popup "Start Auto Cycle" button
	
END_VAR

// ============================================================================
// 0) Default: no request to Auto Cycle unless logic sets it here
// ============================================================================
GVL_HMI.bSystemReady_ReqAutoCycle := FALSE;

// ============================================================================
// 1) Basic "System Ready" condition & Start button blinking
//    - Only blink Start when safety is OK, no incoherence and data loaded
// ============================================================================

// Conditions for "ready to start" as you prefer
IF GVL_Safety.bSafetyEnable
   AND NOT GVL_HMI.bIncoherenceDetected THEN
    bSystemReadyToStart := TRUE;
ELSE
    bSystemReadyToStart := FALSE;
END_IF

// Start button blinking only when system is ready
fbBlinkStartButton(
    bEnable := bSystemReadyToStart,
    tPeriod := T#1S
);
GVL_IO.gDigOutputs.bStartIndicator := fbBlinkStartButton.bBlink;

// ============================================================================
// 2) Handle main Start button on System Ready
//    - Rising edge on Start button
//    - If "ready to start" -> open popup for comment
//    - If not ready / incoherence -> raise alert (same behavior as before)
// ============================================================================

rTrigStartButton(CLK := GVL_IO.gDigInputs.bStartButton);

IF rTrigStartButton.Q THEN
    IF bSystemReadyToStart THEN
        // No incoherence and everything loaded: request popup for comment
        GVL_HMI.bShowAutoCyclePopup   := TRUE;
        GVL_HMI.bIncoherenceAlert     := FALSE;

        // Optionally clear previous comment and reset popup button
        GVL_HMI.sAutoCycleComment     := '';
        GVL_HMI.bStartAutoCycleButton := FALSE;
    ELSE
        // Not ready: keep the "old behavior": show incoherence / warning
        GVL_HMI.bIncoherenceAlert := TRUE;
    END_IF
END_IF

// ============================================================================
// 3) Handle popup "Start Auto Cycle" button
//    - Rising edge on bStartAutoCycleButton
//    - Double-check safety, incoherence and comment length
//    - If OK -> raise bSystemReady_ReqAutoCycle (one-shot)
// ============================================================================

rTrigPopupStartBtn(CLK := GVL_HMI.bStartAutoCycleButton);

IF rTrigPopupStartBtn.Q THEN

    // Extra safety: conditions may have changed since popup was opened
    IF GVL_Safety.bSafetyEnable
       AND NOT GVL_HMI.bIncoherenceDetected
       AND (LEN(GVL_HMI.sAutoCycleComment) > 0) THEN

        // All good: request transition to AUTO_CYCLE
        GVL_HMI.bSystemReady_ReqAutoCycle := TRUE;

        // Close popup
        GVL_HMI.bShowAutoCyclePopup := FALSE;

        // Optionally keep comment for logging

    ELSE
        // Something is wrong:
        // - Safety disabled
        // - Incoherence detected
        // - Or empty comment
        IF GVL_HMI.bIncoherenceDetected THEN
            GVL_HMI.bIncoherenceAlert := TRUE;
        END_IF

        // Reset popup start button, keep popup open so the user can fix it
        GVL_HMI.bStartAutoCycleButton := FALSE;
    END_IF

END_IF

END_PROGRAM

// ---- POUs/Utilities/PRG_UpdateVariablesMoving.TcPOU
PROGRAM PRG_UpdateVariablesMoving
VAR
	bFirstVariablesAssignment  : BOOL := FALSE;
	bValvesSettingsAssignment  : BOOL := FALSE;
	bPumpsFactorAssignment	   : BOOL := FALSE;
	bPumpsSettingsAssignment   : BOOL := FALSE;
	bPumpsDeadVolumeAssignment : BOOL := FALSE;
	
	i : UINT := 1;
	
	aDebug	: ARRAY[1..10] OF BOOL;
	bUpdatePumpFactor	: BOOL := FALSE;
	
END_VAR

IF NOT GVL_IO.gDigInputs.bAccessDoor4InterlockFdbk AND NOT GVL_IO.gDigInputs.bAccessDoor5InterlockFdbk AND NOT GVL_IO.gDigInputs.bAccessDoor6InterlockFdbk THEN
	GVL_Safety.SafetyOutputs.bBelowDoorsFeedback := TRUE;
ELSE
	GVL_Safety.SafetyOutputs.bBelowDoorsFeedback := FALSE;
END_IF

// Mapping bellow doors signals as they are not in safety DI
(*
GVL_IO.gRelayOutputs.bSampleRecoveryLight 		:= NOT GVL_Safety.bTopDoorsClosedFeedback;
GVL_IO.gRelayOutputs.bStageCollectionLeftLight 	:= NOT GVL_Safety.bTopDoorsClosedFeedback;
GVL_IO.gRelayOutputs.bStageCollectionRightLight := NOT GVL_Safety.bTopDoorsClosedFeedback;
*)

// Vial Rack position check
IF GVL_IO.gProfinetInput.iCurrentValue > 120000 THEN
	GVL_IO.bVialRackPresent := TRUE;
ELSE
	GVL_IO.bVialRackPresent := FALSE;
END_IF

// Valves Settings Assignment
IF NOT bValvesSettingsAssignment THEN
	FOR i := 1 TO 5 DO
		GVL_Motion.aValves[i].rTargetVel := 600;
		GVL_Motion.aValves[i].rAcceleration := 200;
		GVL_Motion.aValves[i].rDeceleration := 200;
	END_FOR
	bValvesSettingsAssignment := TRUE;
END_IF

//Pumps factor Assignment [ml/rev]
IF NOT bPumpsFactorAssignment OR bUpdatePumpFactor THEN

	FOR i := 1 TO 10 DO
		GVL_Motion.aPumps[i].Rotary.rPumpFactorFillJars 	:= GVL_Retain.aCalibrationPumpFactor[i];
		GVL_Motion.aPumps[i].Rotary.rPumpFactorFillCalBox 	:= GVL_Retain.aCalibrationPumpFactor[i];
		GVL_Motion.aPumps[i].Rotary.rPumpFactorFromCalBox	:= GVL_Retain.aCalibrationPumpFactor[i];
	END_FOR
		
	bPumpsFactorAssignment := TRUE;
END_IF

//Pumps line dead Volume pipes/tubing Assignment [ml]
IF NOT bPumpsDeadVolumeAssignment THEN
	GVL_Motion.aPumps[1].Rotary.rDeadVolume := -0.3;//4.5;//10.0;
	GVL_Motion.aPumps[2].Rotary.rDeadVolume := -0.5;//8.0;//10.0;
	GVL_Motion.aPumps[3].Rotary.rDeadVolume := 0.65;//5.5;//27.0;
	GVL_Motion.aPumps[4].Rotary.rDeadVolume := 0.2;//6.5;//19.0;
	GVL_Motion.aPumps[5].Rotary.rDeadVolume := 2.3;//10.5;//14.0;
	GVL_Motion.aPumps[6].Rotary.rDeadVolume := 0.65;//7.5;//21.0;
	GVL_Motion.aPumps[7].Rotary.rDeadVolume := 0.85;//8.3;//21.0;
	GVL_Motion.aPumps[8].Rotary.rDeadVolume := -0.3;//6.0;//12.0;
	GVL_Motion.aPumps[9].Rotary.rDeadVolume := 1.4;//7.9;//16.0;
	GVL_Motion.aPumps[10].Rotary.rDeadVolume := 0.8;//8.1;//16.0;
END_IF

//Pumps Settings Assignment
IF NOT bPumpsSettingsAssignment THEN
	FOR i := 1 TO 10 DO
		GVL_Motion.aPumps[i].Rotary.rSpeed := 1800; //1800º/sec with is equal to 300 revs/min
		GVL_Motion.aPumps[i].Rotary.rAcceleration := 2000; //Standard Acceleration based on motor speed
		GVL_Motion.aPumps[i].Rotary.rDeceleration := 2000; //Standard Acceleration based on motor speed
	END_FOR
	bPumpsSettingsAssignment := TRUE;
END_IF

//Pumps Home sensor bit
GVL_Motion.aPumps[1].Linear.bHomeSensorState := GVL_Motion.aPumps[1].Linear.iHomeSensor.0; 
GVL_Motion.aPumps[2].Linear.bHomeSensorState := GVL_Motion.aPumps[2].Linear.iHomeSensor.0; 
GVL_Motion.aPumps[3].Linear.bHomeSensorState := GVL_Motion.aPumps[3].Linear.iHomeSensor.0; 
GVL_Motion.aPumps[4].Linear.bHomeSensorState := GVL_Motion.aPumps[4].Linear.iHomeSensor.0; 
GVL_Motion.aPumps[5].Linear.bHomeSensorState := GVL_Motion.aPumps[5].Linear.iHomeSensor.0; 
GVL_Motion.aPumps[6].Linear.bHomeSensorState := GVL_Motion.aPumps[6].Linear.iHomeSensor.0; 
GVL_Motion.aPumps[7].Linear.bHomeSensorState := GVL_Motion.aPumps[7].Linear.iHomeSensor.0; 
GVL_Motion.aPumps[8].Linear.bHomeSensorState := GVL_Motion.aPumps[8].Linear.iHomeSensor.0; 
GVL_Motion.aPumps[9].Linear.bHomeSensorState := GVL_Motion.aPumps[9].Linear.iHomeSensor.0; 
GVL_Motion.aPumps[10].Linear.bHomeSensorState := GVL_Motion.aPumps[10].Linear.iHomeSensor.0; 

// Pump factor Restore
IF aDebug[1] THEN
	GVL_Retain.aCalibrationPumpFactor[1] := 0.1;
END_IF
IF aDebug[2] THEN
	GVL_Retain.aCalibrationPumpFactor[2] := 0.1;
END_IF
IF aDebug[3] THEN
	GVL_Retain.aCalibrationPumpFactor[3] := 0.1;
END_IF
IF aDebug[4] THEN
	GVL_Retain.aCalibrationPumpFactor[4] := 0.1;
END_IF
IF aDebug[5] THEN
	GVL_Retain.aCalibrationPumpFactor[5] := 0.1;
END_IF
IF aDebug[6] THEN
	GVL_Retain.aCalibrationPumpFactor[6] := 0.1;
END_IF
IF aDebug[7] THEN
	GVL_Retain.aCalibrationPumpFactor[7] := 0.1;
END_IF
IF aDebug[8] THEN
	GVL_Retain.aCalibrationPumpFactor[8] := 0.1;
END_IF
IF aDebug[9] THEN
	GVL_Retain.aCalibrationPumpFactor[9] := 0.1;
END_IF
IF aDebug[10] THEN
	GVL_Retain.aCalibrationPumpFactor[10] := 0.1;
END_IF


// temporary until we are able to get this parameter from hmi or configuration File **************************************************************************
IF NOT bFirstVariablesAssignment THEN
	//Default Homing Motors settings
	GVL_Motion.M1Motor.rHomeAcc 	:= 20.0;
	GVL_Motion.M1Motor.rHomeDec 	:= 20.0;
	GVL_Motion.M1Motor.rHomeVel 	:= 15.0;
	GVL_Motion.M2Motor.rHomeAcc 	:= 20.0;
	GVL_Motion.M2Motor.rHomeDec 	:= 20.0;
	GVL_Motion.M2Motor.rHomeVel 	:= 15.0;
	GVL_Motion.M3Motor.rHomeAcc 	:= 20.0;
	GVL_Motion.M3Motor.rHomeDec 	:= 20.0;
	GVL_Motion.M3Motor.rHomeVel 	:= 15.0;
	
	FOR i :=1 TO 5 DO
		GVL_Motion.aValves[i].rHomeAcc := 400.0;
		GVL_Motion.aValves[i].rHomeDec := 400.0;
		GVL_Motion.aValves[i].rHomeVel := 500.0;
	END_FOR
	
	FOR i :=1 TO 10 DO
		GVL_Motion.aPumps[i].Linear.rHomeAcc := 100.0;
		GVL_Motion.aPumps[i].Linear.rHomeDec := 100.0;
		GVL_Motion.aPumps[i].Linear.rHomeVel := 200.0;
	END_FOR
	
	GVL_Settings.stMachineParam.fM1PositionDeceleration := 30;
	
	bFirstVariablesAssignment := TRUE;
	(*
	GVL_Retain.rLinearPumpOldPosition[1] := -700.0;
	GVL_Retain.rLinearPumpOldPosition[2] := -700.0;
	GVL_Retain.rLinearPumpOldPosition[3] := -700.0;
	GVL_Retain.rLinearPumpOldPosition[4] := -700.0;
	GVL_Retain.rLinearPumpOldPosition[5] := -700.0;
	GVL_Retain.rLinearPumpOldPosition[6] := -700.0;
	GVL_Retain.rLinearPumpOldPosition[7] := -700.0;
	GVL_Retain.rLinearPumpOldPosition[8] := -700.0;
	GVL_Retain.rLinearPumpOldPosition[9] := -700.0;
	GVL_Retain.rLinearPumpOldPosition[10] := -700.0;
	*)
	
END_IF

END_PROGRAM

// ---- POUs/1. MachineControl/PRG_SafetyHandle.TcPOU
PROGRAM PRG_SafetyHandle
VAR
	//Air Supply testing
	bAirSupplyEnable: BOOL	:= TRUE;
	bAirSupplyReset	: BOOL	:= FALSE;
	
	bLockDoors	  	: BOOL 	:= FALSE;	   	// Variable that sends the lock doors signal
	
	tonStabilizingFaults : TON;
	tonClearFaults		 : TON;
	
	i	: USINT;
END_VAR

//Safety Restart & Error Ack
IF GVL_Safety.SafetyInputs.bMachineReset OR GVL_Safety.bM1STOErrorAck THEN
	GVL_Safety.bSafetyErrorAck			:= TRUE;
	GVL_Motion.M1Motor.bTS_ErrorAck		:= TRUE;
ELSE
	GVL_Safety.bSafetyErrorAck			:= FALSE;
	GVL_Motion.M1Motor.bTS_ErrorAck		:= FALSE;
END_IF

GVL_Safety.iM4STOErrorAck			:= GVL_Safety.SafetyInputs.bMachineReset;
GVL_Safety.iM5STOErrorAck			:= GVL_Safety.SafetyInputs.bMachineReset;
GVL_Safety.iM6STOErrorAck			:= GVL_Safety.SafetyInputs.bMachineReset;
GVL_Safety.iM7STOErrorAck			:= GVL_Safety.SafetyInputs.bMachineReset;
GVL_Safety.iM8STOErrorAck			:= GVL_Safety.SafetyInputs.bMachineReset;

GVL_Safety.bSafetyRun				:= TRUE;
GVL_Motion.M1Motor.bTS_Run			:= TRUE;
GVL_Safety.iM4STORun				:= TRUE;
GVL_Safety.iM5STORun				:= TRUE;
GVL_Safety.iM6STORun				:= TRUE;
GVL_Safety.iM7STORun				:= TRUE;
GVL_Safety.iM8STORun				:= TRUE;

IF bAirSupplyEnable THEN
	GVL_Safety.bAirSupplyEnable := TRUE;
ELSE
	GVL_Safety.bAirSupplyEnable	:= FALSE;
END_IF

IF bAirSupplyReset THEN
	GVL_Safety.bAirSupplyReset 	:= TRUE;
ELSE
	GVL_Safety.bAirSupplyReset	:= FALSE;
END_IF

//Alias signal for the reset button blinking
IF GVL_Safety.bResetButtonBlink THEN
	GVL_IO.gDigOutputs.bResetIndicator	:= TRUE;
ELSE
	GVL_IO.gDigOutputs.bResetIndicator	:= FALSE;
END_IF

IF bLockDoors THEN
	GVL_Safety.SafetyOutputs.bLockDoorSafety := TRUE;
	ELSE
	GVL_Safety.SafetyOutputs.bLockDoorSafety := FALSE;
END_IF

// ====================================================================
// 1. SAFETY FAULT LOGIC (STOP & DISABLE ALL PUMPS)
// ====================================================================
// This section executes every PLC cycle while the safety condition is NOT met.

IF NOT GVL_Safety.bSafetyEnable AND GVL_Motion.bInitialHomingDone THEN
	// Immediate Stop and Disable all pumps and linear motors for safety
	FOR i := 1 TO 10 DO
		// 1. Initiate Controlled Stop (MC_Stop) to cancel any active motion commands
		GVL_Motion.aPumpsRotary[i].Stop(); 
		GVL_Motion.aPumpsLinear[i].Stop();
		
		// 2. Immediate Torque Cut-Off (MC_Power.Enable := FALSE)
		GVL_Motion.aPumpsRotary[i].Disable();
		GVL_Motion.aPumpsLinear[i].Disable();
	END_FOR
END_IF

// ====================================================================
// 2. Immediate Fault Command from software conditions
// ====================================================================
// This section activates an immediate fault from alarms flags 

IF GVL_Safety.bSafetyEnable THEN
	GVL_Safety.bImmediateFaultCommand := 
	GVL_Alarms.arrEventFlag[50] OR GVL_Alarms.arrEventFlag[51] OR GVL_Alarms.arrEventFlag[52] OR 
	GVL_Alarms.arrEventFlag[53] OR GVL_Alarms.arrEventFlag[54] OR GVL_Alarms.arrEventFlag[55] OR 
	GVL_Alarms.arrEventFlag[56] OR GVL_Alarms.arrEventFlag[57] OR GVL_Alarms.arrEventFlag[58] OR 
	GVL_Alarms.arrEventFlag[59] OR GVL_Alarms.arrEventFlag[60] OR GVL_Alarms.arrEventFlag[61] OR 
	GVL_Alarms.arrEventFlag[62] OR GVL_Alarms.arrEventFlag[63] OR GVL_Alarms.arrEventFlag[64] OR 
	GVL_Alarms.arrEventFlag[65] OR GVL_Alarms.arrEventFlag[66] OR GVL_Alarms.arrEventFlag[67] OR 
	GVL_Alarms.arrEventFlag[68] OR GVL_Alarms.arrEventFlag[69] OR GVL_Alarms.arrEventFlag[70] OR 
	GVL_Alarms.arrEventFlag[71] OR GVL_Alarms.arrEventFlag[72] OR GVL_Alarms.arrEventFlag[73] OR 
	GVL_Alarms.arrEventFlag[74] OR GVL_Alarms.arrEventFlag[75] OR GVL_Alarms.arrEventFlag[76] OR 
	GVL_Alarms.arrEventFlag[77] OR GVL_Alarms.arrEventFlag[78] OR GVL_Alarms.arrEventFlag[79] OR 
	GVL_Alarms.arrEventFlag[80] OR GVL_Alarms.arrEventFlag[81] OR GVL_Alarms.arrEventFlag[82] OR 
	GVL_Alarms.arrEventFlag[83] OR GVL_Alarms.arrEventFlag[84] OR GVL_Alarms.arrEventFlag[85] OR 
	GVL_Alarms.arrEventFlag[86] OR GVL_Alarms.arrEventFlag[200] OR GVL_Alarms.arrEventFlag[201] OR
	GVL_Alarms.arrEventFlag[202] OR GVL_Alarms.arrEventFlag[203] OR (*GVL_Alarms.arrEventFlag[204] OR*) 
	GVL_Alarms.arrEventFlag[205] OR GVL_Alarms.arrEventFlag[206] OR GVL_Alarms.arrEventFlag[207] OR 
	GVL_Alarms.arrEventFlag[208] OR GVL_Alarms.arrEventFlag[209] OR GVL_Alarms.arrEventFlag[210] OR 
	GVL_Alarms.arrEventFlag[211] OR GVL_Alarms.arrEventFlag[212] OR GVL_Alarms.arrEventFlag[213] OR 
	GVL_Alarms.arrEventFlag[214] OR GVL_Alarms.arrEventFlag[215] OR GVL_Alarms.arrEventFlag[216] OR 
	GVL_Alarms.arrEventFlag[217] OR GVL_Alarms.arrEventFlag[218] OR GVL_Alarms.arrEventFlag[219] OR 
	GVL_Alarms.arrEventFlag[220] OR GVL_Alarms.arrEventFlag[221] OR GVL_Alarms.arrEventFlag[222] OR 
	GVL_Alarms.arrEventFlag[223] OR GVL_Alarms.arrEventFlag[224];
ELSE
	GVL_Safety.bImmediateFaultCommand := FALSE;
END_IF

END_PROGRAM

// ---- POUs/MotionControl/PRG_AxisAssignment.TcPOU
PROGRAM PRG_AxisAssignment
VAR
	bInitDone : BOOL := FALSE;
END_VAR

//Objets Motors Axis Assignment - to use the FB_MotoWrrapper at any part of the software 
IF NOT bInitDone THEN
	
    GVL_Motion.aMotors[1](Axis := GVL_Motion.M1Motor.Axis);				//Motor M1 - Y Axis Stage Collection
    GVL_Motion.aMotors[2](Axis := GVL_Motion.M2Motor.Axis);				//Motor M2 - N Axis Sample Recovery 
	GVL_Motion.aMotors[3](Axis := GVL_Motion.M3Motor.Axis);				//Motor M2 - N Axis Sample Recovery 
	
	GVL_Motion.aPumpsLinear[1](Axis := GVL_Motion.aPumps[1].Linear.Axis);	//Pump 1 - Linear Actuador 
	GVL_Motion.aPumpsLinear[2](Axis := GVL_Motion.aPumps[2].Linear.Axis);	//Pump 2 - Linear Actuador 
	GVL_Motion.aPumpsLinear[3](Axis := GVL_Motion.aPumps[3].Linear.Axis);	//Pump 3 - Linear Actuador 
	GVL_Motion.aPumpsLinear[4](Axis := GVL_Motion.aPumps[4].Linear.Axis);	//Pump 4 - Linear Actuador 
	GVL_Motion.aPumpsLinear[5](Axis := GVL_Motion.aPumps[5].Linear.Axis);	//Pump 5 - Linear Actuador 
	GVL_Motion.aPumpsLinear[6](Axis := GVL_Motion.aPumps[6].Linear.Axis);	//Pump 6 - Linear Actuador 
	GVL_Motion.aPumpsLinear[7](Axis := GVL_Motion.aPumps[7].Linear.Axis);	//Pump 7 - Linear Actuador 
	GVL_Motion.aPumpsLinear[8](Axis := GVL_Motion.aPumps[8].Linear.Axis);	//Pump 8 - Linear Actuador 
	GVL_Motion.aPumpsLinear[9](Axis := GVL_Motion.aPumps[9].Linear.Axis);	//Pump 9 - Linear Actuador 
	GVL_Motion.aPumpsLinear[10](Axis := GVL_Motion.aPumps[10].Linear.Axis);	//Pump 10 - Linear Actuador 
	
	GVL_Motion.aPumpsRotary[1](Axis := GVL_Motion.aPumps[1].Rotary.Axis);	//Pump 1 - Rotary Actuador 
	GVL_Motion.aPumpsRotary[2](Axis := GVL_Motion.aPumps[2].Rotary.Axis);	//Pump 2 - Rotary Actuador 
	GVL_Motion.aPumpsRotary[3](Axis := GVL_Motion.aPumps[3].Rotary.Axis);	//Pump 3 - Rotary Actuador 
	GVL_Motion.aPumpsRotary[4](Axis := GVL_Motion.aPumps[4].Rotary.Axis);	//Pump 4 - Rotary Actuador 
	GVL_Motion.aPumpsRotary[5](Axis := GVL_Motion.aPumps[5].Rotary.Axis);	//Pump 5 - Rotary Actuador 
	GVL_Motion.aPumpsRotary[6](Axis := GVL_Motion.aPumps[6].Rotary.Axis);	//Pump 6 - Rotary Actuador 
	GVL_Motion.aPumpsRotary[7](Axis := GVL_Motion.aPumps[7].Rotary.Axis);	//Pump 7 - Rotary Actuador 
	GVL_Motion.aPumpsRotary[8](Axis := GVL_Motion.aPumps[8].Rotary.Axis);	//Pump 8 - Rotary Actuador 
	GVL_Motion.aPumpsRotary[9](Axis := GVL_Motion.aPumps[9].Rotary.Axis);	//Pump 9 - Rotary Actuador 
	GVL_Motion.aPumpsRotary[10](Axis := GVL_Motion.aPumps[10].Rotary.Axis);	//Pump 10 - Rotary Actuador 
	
	GVL_Motion.aValvesObj[1](Axis := GVL_Motion.aValves[1].Axis);			//Valve 1 - Stepper Motor 
	GVL_Motion.aValvesObj[2](Axis := GVL_Motion.aValves[2].Axis);			//Valve 2 - Stepper Motor 
	GVL_Motion.aValvesObj[3](Axis := GVL_Motion.aValves[3].Axis);			//Valve 3 - Stepper Motor 
	GVL_Motion.aValvesObj[4](Axis := GVL_Motion.aValves[4].Axis);			//Valve 4 - Stepper Motor 
	GVL_Motion.aValvesObj[5](Axis := GVL_Motion.aValves[5].Axis);			//Valve 5 - Stepper Motor 
	
    bInitDone := TRUE;
	
END_IF

END_PROGRAM

// ---- POUs/7. EventsAndAlarms/Marco/POU_EventTest.TcPOU
PROGRAM POU_EventTest
VAR
	fb_EventLog: FB_EventLog;
	
END_VAR



ACT_Event_Mapping(); //Responsable for mapping the events string

// ----- Calling Event Log FB Template ----------------------------------------------------------------------------------------------------

fb_EventLog(bEnable:= TRUE,
			sDateTime:= PRG_MasterSystemTime.sDateTimeSpaces, //Template to generate a date time string (DD.MM.YYYY HH:MM:SS)
			aEventFlags:= GVL_Alarms.arrEventFlag, //Array of bool used to enumerate the events
			aEventTexts:= GVL_Alarms.arrEventText, //Array of string used to descript the events (will be conected with flag array)
			aActiveEvents:= GVL_Alarms.arrActiveEvents, //Array of string used to show the actived events
			aEventLog:= GVL_Alarms.arrEventLogs); //Array of string used to show all FB logs generated

//-----------------------------------------------------------------------------------------------------------------------------------------

ACTION ACT_Event_Mapping:
//--------------------------------
(*
ES -> Emergency Stop
ME -> Motion Error
IE -> Interlock Error
PW -> Process Warning
SF -> System Fault
*)
//----- Emergency Stop ---------------------------------------------------------------------------------------------------------------

GVL_Alarms.arrEventText[0] := 'ES-000: HMI E-Stop Button Active.'; 	//OK
GVL_Alarms.arrEventText[1] := 'ES-001: Side E-Stop Button Active.';	//OK
GVL_Alarms.arrEventText[2] := 'ES-002: Door 1 Open.';	//OK
GVL_Alarms.arrEventText[3] := 'ES-003: Door 2 Open.';	//OK
GVL_Alarms.arrEventText[4] := 'ES-004: Door 3 Open.';	//OK
GVL_Alarms.arrEventText[5] := 'ES-005: Door 4 Open.';	//OK
GVL_Alarms.arrEventText[6] := 'ES-006: Door 5 Open.';	//OK
GVL_Alarms.arrEventText[7] := 'ES-007: Door 6 Open.';	//OK
GVL_Alarms.arrEventText[8] := 'ES-008: Terminal EL6910 FB Error.';	//OK
GVL_Alarms.arrEventText[9] := 'ES-009: Terminal EL6910 Communication Error.';	//OK

//------------------------------------------------------------------------------------------------------------------------------------

//----- Motion Error -----------------------------------------------------------------------------------------------------------------

GVL_Alarms.arrEventText[50] := 'ME-050: Vertical Axis Stage Collection Error.';		//OK
GVL_Alarms.arrEventText[51] := 'ME-051: Vertical Axis Sample Recovery Error.';		//OK
GVL_Alarms.arrEventText[52] := 'ME-052: Horizontal Axis Sample Recovery Error.';	//OK
GVL_Alarms.arrEventText[53] := 'ME-053: Opening Control Pump 1 Motor Error.';		//OK
GVL_Alarms.arrEventText[54] := 'ME-054: Opening Control Pump 2 Motor Error.';		//OK
GVL_Alarms.arrEventText[55] := 'ME-055: Opening Control Pump 3 Motor Error.';		//OK
GVL_Alarms.arrEventText[56] := 'ME-056: Opening Control Pump 4 Motor Error.';		//OK
GVL_Alarms.arrEventText[57] := 'ME-057: Opening Control Pump 5 Motor Error.';		//OK
GVL_Alarms.arrEventText[58] := 'ME-058: Opening Control Pump 6 Motor Error.';		//OK
GVL_Alarms.arrEventText[59] := 'ME-059: Opening Control Pump 7 Motor Error.';		//OK
GVL_Alarms.arrEventText[60] := 'ME-060: Opening Control Pump 8 Motor Error.';		//OK
GVL_Alarms.arrEventText[61] := 'ME-061: Opening Control Pump 9 Motor Error.';		//OK
GVL_Alarms.arrEventText[62] := 'ME-062: Opening Control Pump 10 Motor Error.';		//OK
GVL_Alarms.arrEventText[63] := 'ME-063: Rotary Pump 1 Motor Error.';	//OK
GVL_Alarms.arrEventText[64] := 'ME-064: Rotary Pump 2 Motor Error.';	//OK
GVL_Alarms.arrEventText[65] := 'ME-065: Rotary Pump 3 Motor Error.';	//OK
GVL_Alarms.arrEventText[66] := 'ME-066: Rotary Pump 4 Motor Error.';	//OK
GVL_Alarms.arrEventText[67] := 'ME-067: Rotary Pump 5 Motor Error.';	//OK
GVL_Alarms.arrEventText[68] := 'ME-068: Rotary Pump 6 Motor Error.';	//OK
GVL_Alarms.arrEventText[69] := 'ME-069: Rotary Pump 7 Motor Error.';	//OK
GVL_Alarms.arrEventText[70] := 'ME-070: Rotary Pump 8 Motor Error.';	//OK
GVL_Alarms.arrEventText[71] := 'ME-071: Rotary Pump 9 Motor Error.';	//OK
GVL_Alarms.arrEventText[72] := 'ME-072: Rotary Pump 10 Motor Error.';	//OK
GVL_Alarms.arrEventText[73] := 'ME-073: Valve Motor 1 Error.';	//OK
GVL_Alarms.arrEventText[74] := 'ME-074: Valve Motor 2 Error.';	//OK
GVL_Alarms.arrEventText[75] := 'ME-075: Valve Motor 3 Error.';	//OK
GVL_Alarms.arrEventText[76] := 'ME-076: Valve Motor 4 Error.';	//OK
GVL_Alarms.arrEventText[77] := 'ME-077: Valve Motor 5 Error.';	//OK
GVL_Alarms.arrEventText[78] := 'ME-078: Motion Command Timeout';
GVL_Alarms.arrEventText[79] := 'ME-079: Soft Limit Reached';
GVL_Alarms.arrEventText[80] := 'ME-080: Jog Command Rejected by Interlock';
GVL_Alarms.arrEventText[81] := 'ME-081: Valve Position Mismatch (no in-slot)';
GVL_Alarms.arrEventText[82] := 'ME-082: Axis Emergency Stop Pump Deceleration Active';	//OK
GVL_Alarms.arrEventText[83] := CONCAT('ME-083: System Init Failed - Timeout on Reset ', GVL_Alarms.sMotionResetTimeoutAxis);	//OK
GVL_Alarms.arrEventText[84] := CONCAT('ME-084: System Init Failed - Timeout on Enable ', GVL_Alarms.sMotionEnableTimeoutAxis);	//OK
GVL_Alarms.arrEventText[85] := CONCAT('ME-085: System Init Failed - Timeout on Homing ', GVL_Alarms.sMotionHomeTimeoutAxis);	//OK
GVL_Alarms.arrEventText[86] := CONCAT('ME-086: System Init Failed - Timeout on Motion ', GVL_Alarms.sMotionMoveAbsTimeoutAxis);	//OK

//------------------------------------------------------------------------------------------------------------------------------------

//----- Interlock Error --------------------------------------------------------------------------------------------------------------

GVL_Alarms.arrEventText[100] := 'IE-100: M2 Movement Not allowed';	// OK
GVL_Alarms.arrEventText[101] := 'IE-101: M3 Movement Not allowed';	// OK
GVL_Alarms.arrEventText[102] := 'IE-102: Attempt going Auto Cycle without a Recipe';	//OK
GVL_Alarms.arrEventText[103] := 'IE-103: Attempt going Auto Cycle without Throat stage in correct position';	//OK
GVL_Alarms.arrEventText[104] := 'IE-104: Attempt going Auto Cycle without Vias Rack in correct position';	//OK
GVL_Alarms.arrEventText[105] := 'IE-105: Attempt going Auto Cycle With Solvent 1 Low level';	//OK
GVL_Alarms.arrEventText[106] := 'IE-106: Attempt going Auto Cycle With Solvent 2 Low level';	//OK
GVL_Alarms.arrEventText[107] := 'IE-107: Attempt going Auto Cycle With Solvent 3 Low level';	//OK
GVL_Alarms.arrEventText[108] := 'IE-108: Attempt going Auto Cycle With Solvent 4 Low level';	//OK
GVL_Alarms.arrEventText[109] := 'IE-109: Attempt going Auto Cycle With Waste Bottle high level';	//OK
GVL_Alarms.arrEventText[110] := 'IE-110: Attempt to perform a calibration procedure without a calibration box';	// Need HMI trigger implementation
GVL_Alarms.arrEventText[111] := 'IE-111: M1 Movement Not allowed';	// OK
GVL_Alarms.arrEventText[112] := CONCAT('IE-112: ',GVL_Alarms.sStartCalibrationBlockedReason);


//------------------------------------------------------------------------------------------------------------------------------------

//----- Process Warning --------------------------------------------------------------------------------------------------------------

GVL_Alarms.arrEventText[150] := 'PW-150: Solvent 1 Near Low Level';		//OK
GVL_Alarms.arrEventText[151] := 'PW-151: Solvent 2 Near Low Level';		//OK
GVL_Alarms.arrEventText[152] := 'PW-152: Solvent 3 Near Low Level';		//OK
GVL_Alarms.arrEventText[153] := 'PW-153: Solvent 4 Near Low Level';		//OK
GVL_Alarms.arrEventText[154] := 'PW-154: Waste Bottle Near High Level';	//OK
GVL_Alarms.arrEventText[155] := 'PW-155: Line Pressure Low (pneumatics)'; //Valves missing feedback signals
GVL_Alarms.arrEventText[156] := 'PW-156: Flow Instability Detected ( possible cavitation )';
GVL_Alarms.arrEventText[157] := 'PW-157: Estimated Cycle Time Exceeded ( soft limit )';
GVL_Alarms.arrEventText[158] := 'PW-158: Scale Communication Jitter ( retrying )';
GVL_Alarms.arrEventText[159] := 'PW-159: Calibration Due (time/usage)';
GVL_Alarms.arrEventText[160] := 'PW-160: Recipe Uses Deprecated Field(s)';
GVL_Alarms.arrEventText[161] := 'PW-161: Door Sensor Unstable ( chattering )';
GVL_Alarms.arrEventText[162] := 'PW-162: Profinet Communicaton Error ( Vial Rack pen sensor )';	//OK
GVL_Alarms.arrEventText[163] := 'PW-163: Profinet Vial Rack pen sensor error';	//OK
GVL_Alarms.arrEventText[164] := 'PW-164: Internal Waste Tank Overflow sensor';	//OK
GVL_Alarms.arrEventText[165] := 'PW-165: UPS Replace Battery Activated';	//OK
GVL_Alarms.arrEventText[166] := 'PW-166: UPS Ready Signal drop';	//OK
GVL_Alarms.arrEventText[167] := 'PW-167: Term. 9 EL1809 Dig Input Error';	//OK

//------------------------------------------------------------------------------------------------------------------------------------

//----- System Fault -----------------------------------------------------------------------------------------------------------------

GVL_Alarms.arrEventText[200] := 'SF-200: System Powered Off (PLC on Battery)';	//OK
GVL_Alarms.arrEventText[201] := 'SF-201: EtherCAT Error (bus/offline/STATE)';
GVL_Alarms.arrEventText[202] := 'SF-202: TwinSAFE Fault (EL6910/EL1918/EL2904)';	//OK
GVL_Alarms.arrEventText[203] := 'SF-203: Watchdog Timeout (PLC task overload)';	
GVL_Alarms.arrEventText[204] := 'SF-204: Drive STO Active (M1 - M3 or Valves Motors)';	//OK
GVL_Alarms.arrEventText[205] := 'SF-205: Axis Homing Failed (generic)';
GVL_Alarms.arrEventText[206] := 'SF-206: Axis Following Error';
GVL_Alarms.arrEventText[207] := 'SF-207: Limit Switch Trip (hardware)';
GVL_Alarms.arrEventText[209] := 'SF-209: Pump Motor Overcurrent/Overtemp';
GVL_Alarms.arrEventText[210] := 'SF-210: Air Supply Unit Fault (pressure/enable)'; //Valves missing feedback signals
GVL_Alarms.arrEventText[211] := 'SF-211: Vacuum Leak or Not Achieved (hard limit)';
GVL_Alarms.arrEventText[212] := 'SF-212: Scale Communication Error - TCP Connect'; 				//OK
GVL_Alarms.arrEventText[213] := 'SF-213: Scale Communication Error - TCP Send Message';			//OK
GVL_Alarms.arrEventText[214] := 'SF-214: Scale Communication Error - TCP Receive Message';		//OK
GVL_Alarms.arrEventText[215] := 'SF-215: Scale Communication Error - TCP Close Communication';	//OK
GVL_Alarms.arrEventText[216] := 'SF-216: Recipe Load Failed (checksum/version)';
GVL_Alarms.arrEventText[217] := 'SF-217: Data Save Failed (I/O)';
GVL_Alarms.arrEventText[218] := 'SF-218: Disk Space Critically Low';
GVL_Alarms.arrEventText[219] := 'SF-219: NTP/Clock Large Time Jump Detected';
GVL_Alarms.arrEventText[220] := 'SF-220: HMI-PLC Heartbeat Lost';
GVL_Alarms.arrEventText[221] := 'SF-222: Analog Sensor Out-of-Range (broken wire?)';
GVL_Alarms.arrEventText[222] := 'SF-223: DC Invalid Sync Configuration (EtherCAT)';
GVL_Alarms.arrEventText[223] := 'SF-224: Safety Reset Failed';
GVL_Alarms.arrEventText[224] := 'SF-225: Unauthorized User Action Blocked';

//------------------------------------------------------------------------------------------------------------------------------------

//----- Process Fails --------------------------------------------------------------------------------------------------------------

// AUTO CYCLE
GVL_Alarms.arrEventText[300] := 'SF-300: AUTO CYLE - Sealing Failure';
GVL_Alarms.arrEventText[301] := 'SF-301: AUTO CYLE - LeakTest Failure';
GVL_Alarms.arrEventText[302] := 'SF-302: AUTO CYLE - Recovery Failure';
GVL_Alarms.arrEventText[303] := 'SF-303: AUTO CYLE - Washing Failure';
GVL_Alarms.arrEventText[304] := 'SF-304: AUTO CYLE - Drying Failure';
GVL_Alarms.arrEventText[305] := 'SF-305: AUTO CYLE - Auto Cycled Aborted';
GVL_Alarms.arrEventText[306] := 'SF-306: AUTO CYLE - Auto Cycled Stopped';

// CALIBRATION
GVL_Alarms.arrEventText[320] := 'SF-320: CALIBRATION - LeakTest Failure';
GVL_Alarms.arrEventText[321] := 'SF-321: CALIBRATION - Calibration Aborted by Operator';
GVL_Alarms.arrEventText[322] := 'SF-322: CALIBRATION - Calibration Aborted due error';
GVL_Alarms.arrEventText[323] := CONCAT('SF-323: CALIBRATION - Calibration JSON File creation Error, ErrorID: ',TO_STRING(GVL_Alarms.nCalJsonCreationErrorId)); 	//OK

// MANUAL
GVL_Alarms.arrEventText[340] := 'SF-340: MANUAL - Stage Collection Motor Move Timeout';
GVL_Alarms.arrEventText[341] := 'SF-341: MANUAL - Sample Recovery Vertical Motor Move Timeout';
GVL_Alarms.arrEventText[342] := 'SF-342: MANUAL - Sample Recovery Horizontal Motor Move Timeout';
GVL_Alarms.arrEventText[343] := 'SF-343: MANUAL - Valves Movement Timeout';
GVL_Alarms.arrEventText[344] := 'SF-344: MANUAL - Rotary Pumps Move Timeout';

// RECIPE
GVL_Alarms.arrEventText[350] := 'SF-350: RECIPE - Error Loading Recipe';
GVL_Alarms.arrEventText[351] := 'SF-351: RECIPE - Error Saving Recipe';
GVL_Alarms.arrEventText[352] := 'SF-352: RECIPE - Error Editing Recipe';
GVL_Alarms.arrEventText[353] := 'SF-353: RECIPE - Error Activating Recipe';

//------------------------------------------------------------------------------------------------------------------------------------
END_ACTION

END_PROGRAM

// ---- POUs/7. EventsAndAlarms/Marco/PRG_MasterSystemTime.TcPOU
PROGRAM PRG_MasterSystemTime
VAR
	//Variables
	bReadyToRead				:BOOL;
	bFirstScan					:BOOL := TRUE;
	bUpdateSysTime				:BOOL; //Output of pulse generator
	tSysTimeUpdatePeriod		:TIME := T#5S;
	stTimeStamp					:TIMESTRUCT;
	stNullTimeStamp				:TIMESTRUCT;
	sRawDateTime				:STRING;
	sSystemDate					:STRING;
	sSystemTime					:STRING;
	sDateTime					:STRING;
	sDateTimeSpaces				:STRING;
	
	//Functions
	fbGetSystemTime				:TC2_Utilities.NT_GetTime;
	fbRTClock					:TC2_Utilities.RTC_EX2;		//Local real-time clock
	tonTimeUpdateGen			:TC2_Utilities.TON;			//Pulse generator for triggering fbGetSystemTime function
	rtrigSysTimeCollected		:TC2_Utilities.R_TRIG;		//System time collected

END_VAR

//Aux functions call
tonTimeUpdateGen(	IN := NOT bUpdateSysTime,
					PT := tSysTimeUpdatePeriod,
					Q => bUpdateSysTime);

//Get Current System Time
fbGetSystemTime(NETID := ,
				START := bFirstScan OR bUpdateSysTime,
				TMOUT := ,
				BUSY => ,
				ERR => ,
				ERRID => ,
				TIMESTR => );
				
//Get system time done detection - one-shot
rtrigSysTimeCollected(CLK := NOT fbGetSystemTime.BUSY);

//Synchronize Real-Time clock with system time
fbRTClock(	EN := rtrigSysTimeCollected.Q, 
			PDT := fbGetSystemTime.TIMESTR,
			CDT => stTimeStamp, 
			Q => bReadyToRead);

// System Date and Time in Proper Order 
IF bReadyToRead THEN
	sRawDateTime := SYSTEMTIME_TO_STRING(stTimeStamp);  // format: YYYY-MM-DD-hh:mm:ss.xxx
	sSystemDate := CONCAT(CONCAT(CONCAT(CONCAT(MID(sRawDateTime, 2, 9), '.'),  MID(sRawDateTime, 2, 6)), '.'), LEFT(sRawDateTime, 4));
	sSystemTime := MID(sRawDateTime, 8, 12);
	sDateTime := CONCAT(CONCAT(sSystemDate, '  '), sSystemTime);
	sDateTimeSpaces	:= CONCAT(sDateTime, '    ');
END_IF;

bFirstScan := FALSE;

END_PROGRAM

// ---- POUs/7. EventsAndAlarms/Marco/POU_FaultHandler.TcPOU
PROGRAM POU_FaultHandler
VAR
	tonSF200Delay 	: TON;
	bSF200Alarm		: BOOL := FALSE;
END_VAR



//------__________________________----------------------------------------------------------------------------------------------------
//----- Related to Emergency Stop ----------------------------------------------------------------------------------------------------


(*-ES-000: HMI E-Stop Button Active-*)
IF NOT GVL_Safety.SafetyInputs.bEStopHMICh1 OR 
	NOT GVL_Safety.SafetyInputs.bEStopHMICh2 THEN
		GVL_Alarms.arrEventFlag[0]:= TRUE;
	ELSIF GVL_Safety.SafetyInputs.bMachineReset THEN
		GVL_Alarms.arrEventFlag[0]:= FALSE;	
END_IF

(*-ES-001: Side E-Stop Button Active-*)
IF NOT GVL_Safety.SafetyInputs.bEStopSideCh1 OR 
	NOT GVL_Safety.SafetyInputs.bEStopSideCh2 THEN
		GVL_Alarms.arrEventFlag[1]:= TRUE;
	ELSIF GVL_Safety.SafetyInputs.bMachineReset THEN
		GVL_Alarms.arrEventFlag[1]:= FALSE;	
END_IF

(*-ES-002: Door 1 Open-*)
IF NOT GVL_Safety.SafetyInputs.bStageCollectLeftDoorCh1 OR 
	NOT GVL_Safety.SafetyInputs.bStageCollectLeftDoorCh2 THEN
		GVL_Alarms.arrEventFlag[2]:= TRUE;
	ELSIF GVL_Safety.SafetyInputs.bMachineReset THEN
		GVL_Alarms.arrEventFlag[2]:= FALSE;	
END_IF

(*-ES-003: Door 2 Open-*)
IF NOT GVL_Safety.SafetyInputs.bStageCollectRightDoorCh1 OR 
	NOT GVL_Safety.SafetyInputs.bStageCollectRightDoorCh2 THEN
		GVL_Alarms.arrEventFlag[3]:= TRUE;
	ELSIF GVL_Safety.SafetyInputs.bMachineReset THEN
		GVL_Alarms.arrEventFlag[3]:= FALSE;	
END_IF

(*-ES-004: Door 3 Open-*)
IF NOT GVL_Safety.SafetyInputs.bSampleRecoveryDoorCh1 OR 
	NOT GVL_Safety.SafetyInputs.bSampleRecoveryDoorCh2 THEN
		GVL_Alarms.arrEventFlag[4]:= TRUE;
	ELSIF GVL_Safety.SafetyInputs.bMachineReset THEN
		GVL_Alarms.arrEventFlag[4]:= FALSE;	
END_IF

(*-ES-005: Door 4 Open-*)
IF GVL_Safety.SafetyInputs.bD4AccessDoorIntlckOSSD1 OR 
	GVL_Safety.SafetyInputs.bD4AccessDoorIntlckOSSD2 THEN
		GVL_Alarms.arrEventFlag[5]:= TRUE;
	ELSIF GVL_Safety.SafetyInputs.bMachineReset THEN
		GVL_Alarms.arrEventFlag[5]:= FALSE;	
END_IF

(*-ES-006: Door 5 Open-*)
IF GVL_Safety.SafetyInputs.bD5AccessDoorIntlckOSSD1 OR 
	GVL_Safety.SafetyInputs.bD5AccessDoorIntlckOSSD2 THEN
		GVL_Alarms.arrEventFlag[6]:= TRUE;
	ELSIF GVL_Safety.SafetyInputs.bMachineReset THEN
		GVL_Alarms.arrEventFlag[6]:= FALSE;	
END_IF

(*-ES-007: Door 6 Open-*)
IF GVL_Safety.SafetyInputs.bD6AccessDoorIntlckOSSD1 OR 
	GVL_Safety.SafetyInputs.bD6AccessDoorIntlckOSSD2 THEN
		GVL_Alarms.arrEventFlag[7]:= TRUE;
	ELSIF GVL_Safety.SafetyInputs.bMachineReset THEN
		GVL_Alarms.arrEventFlag[7]:= FALSE;	
END_IF

(*-ES-008: Terminal EL6910 FB Error-*)
IF GVL_Safety.SafetyInputs.iSafetyFBError THEN
		GVL_Alarms.arrEventFlag[8]:= TRUE;
	ELSIF GVL_Safety.SafetyInputs.bMachineReset THEN
		GVL_Alarms.arrEventFlag[8]:= FALSE;	
END_IF

(*-ES-009: Terminal EL6910 Communication Error-*)
IF GVL_Safety.SafetyInputs.iSafetyComError THEN
		GVL_Alarms.arrEventFlag[9]:= TRUE;
	ELSIF GVL_Safety.SafetyInputs.bMachineReset THEN
		GVL_Alarms.arrEventFlag[9]:= FALSE;	
END_IF

//*********************************************************END SECTION****************************************************************

//------_________________________-----------------------------------------------------------------------------------------------------
//----- Related to Motion Errors -----------------------------------------------------------------------------------------------------


(*-ME-050: Vertical Axis Stage Collection Error-*)
IF GVL_Motion.M1Motor.iError AND GVL_Safety.bSafetyEnable THEN
		GVL_Alarms.arrEventFlag[50]:= TRUE;
	ELSIF GVL_Safety.SafetyInputs.bMachineReset THEN
		GVL_Alarms.arrEventFlag[50]:= FALSE;	
END_IF

(*-ME-051: Vertical Axis Sample Recovery Error-*)
IF GVL_Motion.M2Motor.iError AND GVL_Safety.bSafetyEnable THEN
		GVL_Alarms.arrEventFlag[51]:= TRUE;
	ELSIF GVL_Safety.SafetyInputs.bMachineReset THEN
		GVL_Alarms.arrEventFlag[51]:= FALSE;	
END_IF

(*-ME-052: Horizontal Axis Sample Recovery Error-*)
IF GVL_Motion.M3Motor.iError AND GVL_Safety.bSafetyEnable THEN
		GVL_Alarms.arrEventFlag[52]:= TRUE;
	ELSIF GVL_Safety.SafetyInputs.bMachineReset THEN
		GVL_Alarms.arrEventFlag[52]:= FALSE;	
END_IF

(*-ME-053: Opening Control Pump 1 Error-*)
IF GVL_Motion.aPumps[1].Linear.iError AND GVL_Safety.bSafetyEnable THEN
		GVL_Alarms.arrEventFlag[53]:= TRUE;
	ELSIF GVL_Safety.SafetyInputs.bMachineReset THEN
		GVL_Alarms.arrEventFlag[53]:= FALSE;	
END_IF

(*-ME-054: Opening Control Pump 2 Error-*)
IF GVL_Motion.aPumps[2].Linear.iError AND GVL_Safety.bSafetyEnable THEN
		GVL_Alarms.arrEventFlag[54]:= TRUE;
	ELSIF GVL_Safety.SafetyInputs.bMachineReset THEN
		GVL_Alarms.arrEventFlag[54]:= FALSE;	
END_IF

(*-ME-055: Opening Control Pump 3 Error-*)
IF GVL_Motion.aPumps[3].Linear.iError AND GVL_Safety.bSafetyEnable THEN
		GVL_Alarms.arrEventFlag[55]:= TRUE;
	ELSIF GVL_Safety.SafetyInputs.bMachineReset THEN
		GVL_Alarms.arrEventFlag[55]:= FALSE;	
END_IF

(*-ME-056: Opening Control Pump 4 Error-*)
IF GVL_Motion.aPumps[4].Linear.iError AND GVL_Safety.bSafetyEnable THEN
		GVL_Alarms.arrEventFlag[56]:= TRUE;
	ELSIF GVL_Safety.SafetyInputs.bMachineReset THEN
		GVL_Alarms.arrEventFlag[56]:= FALSE;	
END_IF

(*-ME-057: Opening Control Pump 5 Error-*)
IF GVL_Motion.aPumps[5].Linear.iError AND GVL_Safety.bSafetyEnable THEN
		GVL_Alarms.arrEventFlag[57]:= TRUE;
	ELSIF GVL_Safety.SafetyInputs.bMachineReset THEN
		GVL_Alarms.arrEventFlag[57]:= FALSE;	
END_IF

(*-ME-058: Opening Control Pump 6 Error-*)
IF GVL_Motion.aPumps[6].Linear.iError AND GVL_Safety.bSafetyEnable THEN
		GVL_Alarms.arrEventFlag[58]:= TRUE;
	ELSIF GVL_Safety.SafetyInputs.bMachineReset THEN
		GVL_Alarms.arrEventFlag[58]:= FALSE;	
END_IF

(*-ME-059: Opening Control Pump 7 Error-*)
IF GVL_Motion.aPumps[7].Linear.iError AND GVL_Safety.bSafetyEnable THEN
		GVL_Alarms.arrEventFlag[59]:= TRUE;
	ELSIF GVL_Safety.SafetyInputs.bMachineReset THEN
		GVL_Alarms.arrEventFlag[59]:= FALSE;	
END_IF

(*-ME-060: Opening Control Pump 8 Error-*)
IF GVL_Motion.aPumps[8].Linear.iError AND GVL_Safety.bSafetyEnable THEN
		GVL_Alarms.arrEventFlag[60]:= TRUE;
	ELSIF GVL_Safety.SafetyInputs.bMachineReset THEN
		GVL_Alarms.arrEventFlag[60]:= FALSE;	
END_IF

(*-ME-061: Opening Control Pump 9 Error-*)
IF GVL_Motion.aPumps[9].Linear.iError AND GVL_Safety.bSafetyEnable THEN
		GVL_Alarms.arrEventFlag[61]:= TRUE;
	ELSIF GVL_Safety.SafetyInputs.bMachineReset THEN
		GVL_Alarms.arrEventFlag[61]:= FALSE;	
END_IF

(*-ME-062: Opening Control Pump 10 Error-*)
IF GVL_Motion.aPumps[10].Linear.iError AND GVL_Safety.bSafetyEnable THEN
		GVL_Alarms.arrEventFlag[62]:= TRUE;
	ELSIF GVL_Safety.SafetyInputs.bMachineReset THEN
		GVL_Alarms.arrEventFlag[62]:= FALSE;	
END_IF

(*-ME-063: Pump Motor 1 Error-*)
IF GVL_Motion.aPumps[1].Rotary.iError AND GVL_Safety.bSafetyEnable THEN
		GVL_Alarms.arrEventFlag[63]:= TRUE;
	ELSIF GVL_Safety.SafetyInputs.bMachineReset THEN
		GVL_Alarms.arrEventFlag[63]:= FALSE;	
END_IF

(*-ME-064: Pump Motor 2 Error-*)
IF GVL_Motion.aPumps[2].Rotary.iError AND GVL_Safety.bSafetyEnable THEN
		GVL_Alarms.arrEventFlag[64]:= TRUE;
	ELSIF GVL_Safety.SafetyInputs.bMachineReset THEN
		GVL_Alarms.arrEventFlag[64]:= FALSE;	
END_IF

(*-ME-065: Pump Motor 3 Error-*)
IF GVL_Motion.aPumps[3].Rotary.iError AND GVL_Safety.bSafetyEnable THEN
		GVL_Alarms.arrEventFlag[65]:= TRUE;
	ELSIF GVL_Safety.SafetyInputs.bMachineReset THEN
		GVL_Alarms.arrEventFlag[65]:= FALSE;	
END_IF

(*-ME-066: Pump Motor 4 Error-*)
IF GVL_Motion.aPumps[4].Rotary.iError AND GVL_Safety.bSafetyEnable THEN
		GVL_Alarms.arrEventFlag[66]:= TRUE;
	ELSIF GVL_Safety.SafetyInputs.bMachineReset THEN
		GVL_Alarms.arrEventFlag[66]:= FALSE;	
END_IF

(*-ME-067: Pump Motor 5 Error-*)
IF GVL_Motion.aPumps[5].Rotary.iError AND GVL_Safety.bSafetyEnable THEN
		GVL_Alarms.arrEventFlag[67]:= TRUE;
	ELSIF GVL_Safety.SafetyInputs.bMachineReset THEN
		GVL_Alarms.arrEventFlag[67]:= FALSE;	
END_IF

(*-ME-068: Pump Motor 6 Error-*)
IF GVL_Motion.aPumps[6].Rotary.iError AND GVL_Safety.bSafetyEnable THEN
		GVL_Alarms.arrEventFlag[68]:= TRUE;
	ELSIF GVL_Safety.SafetyInputs.bMachineReset THEN
		GVL_Alarms.arrEventFlag[68]:= FALSE;	
END_IF

(*-ME-069: Pump Motor 7 Error-*)
IF GVL_Motion.aPumps[7].Rotary.iError AND GVL_Safety.bSafetyEnable THEN
		GVL_Alarms.arrEventFlag[69]:= TRUE;
	ELSIF GVL_Safety.SafetyInputs.bMachineReset THEN
		GVL_Alarms.arrEventFlag[69]:= FALSE;	
END_IF

(*-ME-070: Pump Motor 8 Error-*)
IF GVL_Motion.aPumps[8].Rotary.iError AND GVL_Safety.bSafetyEnable THEN
		GVL_Alarms.arrEventFlag[70]:= TRUE;
	ELSIF GVL_Safety.SafetyInputs.bMachineReset THEN
		GVL_Alarms.arrEventFlag[70]:= FALSE;	
END_IF

(*-ME-071: Pump Motor 9 Error-*)
IF GVL_Motion.aPumps[9].Rotary.iError AND GVL_Safety.bSafetyEnable THEN
		GVL_Alarms.arrEventFlag[71]:= TRUE;
	ELSIF GVL_Safety.SafetyInputs.bMachineReset THEN
		GVL_Alarms.arrEventFlag[71]:= FALSE;	
END_IF

(*-ME-072: Pump Motor 10 Error-*)
IF GVL_Motion.aPumps[10].Rotary.iError AND GVL_Safety.bSafetyEnable THEN
		GVL_Alarms.arrEventFlag[72]:= TRUE;
	ELSIF GVL_Safety.SafetyInputs.bMachineReset THEN
		GVL_Alarms.arrEventFlag[72]:= FALSE;	
END_IF

(*-ME-073: Valve Motor 1 Error-*)
IF GVL_Motion.aValves[1].iError AND GVL_Safety.bSafetyEnable THEN
		GVL_Alarms.arrEventFlag[73]:= TRUE;
	ELSIF GVL_Safety.SafetyInputs.bMachineReset THEN
		GVL_Alarms.arrEventFlag[73]:= FALSE;	
END_IF

(*-ME-074: Valve Motor 2 Error-*)
IF GVL_Motion.aValves[2].iError AND GVL_Safety.bSafetyEnable THEN
		GVL_Alarms.arrEventFlag[74]:= TRUE;
	ELSIF GVL_Safety.SafetyInputs.bMachineReset THEN
		GVL_Alarms.arrEventFlag[74]:= FALSE;	
END_IF

(*-ME-075: Valve Motor 3 Error-*)
IF GVL_Motion.aValves[3].iError AND GVL_Safety.bSafetyEnable THEN
		GVL_Alarms.arrEventFlag[75]:= TRUE;
	ELSIF GVL_Safety.SafetyInputs.bMachineReset THEN
		GVL_Alarms.arrEventFlag[75]:= FALSE;	
END_IF

(*-ME-076: Valve Motor 4 Error-*)
IF GVL_Motion.aValves[4].iError AND GVL_Safety.bSafetyEnable THEN
		GVL_Alarms.arrEventFlag[76]:= TRUE;
	ELSIF GVL_Safety.SafetyInputs.bMachineReset THEN
		GVL_Alarms.arrEventFlag[76]:= FALSE;	
END_IF

(*-ME-077: Valve Motor 5 Error-*)
IF GVL_Motion.aValves[5].iError AND GVL_Safety.bSafetyEnable THEN
		GVL_Alarms.arrEventFlag[77]:= TRUE;
	ELSIF GVL_Safety.SafetyInputs.bMachineReset THEN
		GVL_Alarms.arrEventFlag[77]:= FALSE;	
END_IF


(*-ME-082: Axis Emergency Stop Pump Deceleration Active-*)
IF GVL_Motion.bAnyPumpRunning AND NOT GVL_Safety.bSafetyEnable THEN
		GVL_Alarms.arrEventFlag[82]:= TRUE;
	ELSIF GVL_Safety.SafetyInputs.bMachineReset THEN
		GVL_Alarms.arrEventFlag[82]:= FALSE;	
END_IF

(* ME-083: System Init Failed - Timeout on Reset *)
IF GVL_Alarms.bMotionResetTimeout THEN
		GVL_Alarms.arrEventFlag[83]:= TRUE;
	ELSIF GVL_Safety.SafetyInputs.bMachineReset THEN
		GVL_Alarms.arrEventFlag[83]:= FALSE;	
END_IF

(* ME-084: System Init Failed - Timeout on Enable *)
IF GVL_Alarms.bMotionEnableTimeout THEN
		GVL_Alarms.arrEventFlag[84]:= TRUE;
	ELSIF GVL_Safety.SafetyInputs.bMachineReset THEN
		GVL_Alarms.arrEventFlag[84]:= FALSE;	
END_IF

(* ME-085: System Init Failed - Timeout on Homing *)
IF GVL_Alarms.bMotionHomeTimeout THEN
		GVL_Alarms.arrEventFlag[85]:= TRUE;
	ELSIF GVL_Safety.SafetyInputs.bMachineReset THEN
		GVL_Alarms.arrEventFlag[85]:= FALSE;	
END_IF

(* ME-086: System Init Failed - Timeout on Motion *)
IF GVL_Alarms.bMotionMoveAbsTimeout THEN
		GVL_Alarms.arrEventFlag[86]:= TRUE;
	ELSIF GVL_Safety.SafetyInputs.bMachineReset THEN
		GVL_Alarms.arrEventFlag[86]:= FALSE;	
END_IF

//*********************************************************END SECTION****************************************************************

//------____________________________--------------------------------------------------------------------------------------------------
//----- Related to Interlock Errors --------------------------------------------------------------------------------------------------

(* IE-100: M2 Movement NOT allowed *)
IF GVL_HMI.bM2MoveNotAllowedTrigger THEN
		GVL_Alarms.arrEventFlag[100]:= TRUE;
	ELSIF GVL_Safety.SafetyInputs.bMachineReset THEN
		GVL_Alarms.arrEventFlag[100]:= FALSE;	
END_IF

(* IE-101: M3 Movement Not allowed *)
IF GVL_HMI.bM2MoveNotAllowedTrigger THEN
		GVL_Alarms.arrEventFlag[101]:= TRUE;
	ELSIF GVL_Safety.SafetyInputs.bMachineReset THEN
		GVL_Alarms.arrEventFlag[101]:= FALSE;	
END_IF

(* IE-102: Attempt going Auto Cycle without a Recipe *)
IF GVL_HMI.bIncoherenceAlert AND NOT GVL_Recipe.bIsThereRecipeActivated THEN
		GVL_Alarms.arrEventFlag[102]:= TRUE;
	ELSIF GVL_Safety.SafetyInputs.bMachineReset THEN
		GVL_Alarms.arrEventFlag[102]:= FALSE;	
END_IF

(* IE-103: Attempt going Auto Cycle without Throat stage in correct position *)
IF GVL_HMI.bIncoherenceAlert AND NOT GVL_IO.gDigInputs.bThroatJigPresent THEN
		GVL_Alarms.arrEventFlag[103]:= TRUE;
	ELSIF GVL_Safety.SafetyInputs.bMachineReset THEN
		GVL_Alarms.arrEventFlag[103]:= FALSE;	
END_IF

(* IE-104: Attempt going Auto Cycle without Vias Rack in correct position *)
IF GVL_HMI.bIncoherenceAlert AND NOT GVL_IO.bVialRackPresent THEN
		GVL_Alarms.arrEventFlag[104]:= TRUE;
	ELSIF GVL_Safety.SafetyInputs.bMachineReset THEN
		GVL_Alarms.arrEventFlag[104]:= FALSE;	
END_IF

(* IE-105: Attempt going Auto Cycle With Solvent 1 Low level *)

IF GVL_HMI.bIncoherenceAlert AND GVL_Alarms.aSolventLowLevel[1] THEN
		GVL_Alarms.arrEventFlag[105]:= TRUE;
	ELSIF GVL_Safety.SafetyInputs.bMachineReset THEN
		GVL_Alarms.arrEventFlag[105]:= FALSE;	
END_IF

(* IE-106: Attempt going Auto Cycle With Solvent 2 Low level *)
IF GVL_HMI.bIncoherenceAlert AND GVL_Alarms.aSolventLowLevel[2] THEN
		GVL_Alarms.arrEventFlag[106]:= TRUE;
	ELSIF GVL_Safety.SafetyInputs.bMachineReset THEN
		GVL_Alarms.arrEventFlag[106]:= FALSE;	
END_IF

(* IE-107: Attempt going Auto Cycle With Solvent 3 Low level *)
IF GVL_HMI.bIncoherenceAlert AND GVL_Alarms.aSolventLowLevel[3] THEN
		GVL_Alarms.arrEventFlag[107]:= TRUE;
	ELSIF GVL_Safety.SafetyInputs.bMachineReset THEN
		GVL_Alarms.arrEventFlag[107]:= FALSE;	
END_IF

(* IE-108: Attempt going Auto Cycle With Solvent 4 Low level *)
IF GVL_HMI.bIncoherenceAlert AND GVL_Alarms.aSolventLowLevel[4] THEN
		GVL_Alarms.arrEventFlag[108]:= TRUE;
	ELSIF GVL_Safety.SafetyInputs.bMachineReset THEN
		GVL_Alarms.arrEventFlag[108]:= FALSE;	
END_IF

(* IE-109: Attempt going Auto Cycle With Waste Bottle high level *)
IF GVL_HMI.bIncoherenceAlert AND GVL_Alarms.bWasteHighLevel THEN
		GVL_Alarms.arrEventFlag[109]:= TRUE;
	ELSIF GVL_Safety.SafetyInputs.bMachineReset THEN
		GVL_Alarms.arrEventFlag[109]:= FALSE;	
END_IF

(* IE-110: Attempt to perform a calibration procedure without a calibration box *)
IF GVL_HMI.bCalNotAllowedTrigger THEN
		GVL_Alarms.arrEventFlag[110]:= TRUE;
	ELSIF GVL_Safety.SafetyInputs.bMachineReset THEN
		GVL_Alarms.arrEventFlag[110]:= FALSE;	
END_IF

(* IE-111: M1 Movement Not allowed *)
IF GVL_HMI.bM1MoveNotAllowedTrigger THEN
		GVL_Alarms.arrEventFlag[111]:= TRUE;
	ELSIF GVL_Safety.SafetyInputs.bMachineReset THEN
		GVL_Alarms.arrEventFlag[111]:= FALSE;	
END_IF

(* IE-112: Calibration Solvent Selection *)
IF GVL_Alarms.bInvalidSolventSelection THEN
		GVL_Alarms.arrEventFlag[112]:= TRUE;
	ELSIF GVL_Safety.SafetyInputs.bMachineReset THEN
		GVL_Alarms.arrEventFlag[112]:= FALSE;	
END_IF


//*********************************************************END SECTION****************************************************************

//------____________________________--------------------------------------------------------------------------------------------------
//----- Related to Process Warnings --------------------------------------------------------------------------------------------------

(* PW-150: Solvent 1 Near Low Level *)
IF GVL_Alarms.aSolventNearLowLevel[1] THEN
		GVL_Alarms.arrEventFlag[150]:= TRUE;
	ELSIF GVL_Safety.SafetyInputs.bMachineReset THEN
		GVL_Alarms.arrEventFlag[150]:= FALSE;	
END_IF

(* PW-151: Solvent 2 Near Low Level *)
IF GVL_Alarms.aSolventNearLowLevel[2] THEN
		GVL_Alarms.arrEventFlag[151]:= TRUE;
	ELSIF GVL_Safety.SafetyInputs.bMachineReset THEN
		GVL_Alarms.arrEventFlag[151]:= FALSE;	
END_IF

(* PW-152: Solvent 3 Near Low Level *)
IF GVL_Alarms.aSolventNearLowLevel[3] THEN
		GVL_Alarms.arrEventFlag[152]:= TRUE;
	ELSIF GVL_Safety.SafetyInputs.bMachineReset THEN
		GVL_Alarms.arrEventFlag[152]:= FALSE;	
END_IF

(* PW-153: Solvent 4 Near Low Level *)
IF GVL_Alarms.aSolventNearLowLevel[4] THEN
		GVL_Alarms.arrEventFlag[153]:= TRUE;
	ELSIF GVL_Safety.SafetyInputs.bMachineReset THEN
		GVL_Alarms.arrEventFlag[153]:= FALSE;	
END_IF

(* PW-154: Waste Bottle Near High Level *)
IF GVL_Alarms.bWasteNearHighLevel THEN
		GVL_Alarms.arrEventFlag[154]:= TRUE;
	ELSIF GVL_Safety.SafetyInputs.bMachineReset THEN
		GVL_Alarms.arrEventFlag[154]:= FALSE;	
END_IF

(* PW-162: Profinet Communicaton Error ( Vial Rack pen sensor ) *)
IF GVL_IO.gProfinetInput.iPnIoBoxState <> 0 THEN
		GVL_Alarms.arrEventFlag[162]:= TRUE;
	ELSIF GVL_Safety.SafetyInputs.bMachineReset THEN
		GVL_Alarms.arrEventFlag[162]:= FALSE;	
END_IF

(* PW-163: Profinet Vial Rack pen sensor error *)
IF GVL_IO.gProfinetInput.bErrorStatus THEN
		GVL_Alarms.arrEventFlag[163]:= TRUE;
	ELSIF GVL_Safety.SafetyInputs.bMachineReset THEN
		GVL_Alarms.arrEventFlag[163]:= FALSE;	
END_IF

(* PW-163: Internal Waste Tank Overflow sensor *)
IF GVL_IO.gDigInputs.bWasteOverflowSensor THEN
		GVL_Alarms.arrEventFlag[164]:= TRUE;
	ELSIF GVL_Safety.SafetyInputs.bMachineReset THEN
		GVL_Alarms.arrEventFlag[164]:= FALSE;	
END_IF

(* PW-164: UPS Replace Battery Activated *)
IF GVL_IO.gDigInputs.bUPSReplaceBattery THEN
		GVL_Alarms.arrEventFlag[165]:= TRUE;
	ELSIF GVL_Safety.SafetyInputs.bMachineReset THEN
		GVL_Alarms.arrEventFlag[165]:= FALSE;	
END_IF

(* PW-165: UPS Ready Signal drop *)
IF NOT GVL_IO.gDigInputs.bUPSReady THEN
		GVL_Alarms.arrEventFlag[166]:= TRUE;
	ELSIF GVL_Safety.SafetyInputs.bMachineReset THEN
		GVL_Alarms.arrEventFlag[166]:= FALSE;	
END_IF

(*PW-167: Term. 9 EL1809 Dig Input Error*)
IF GVL_IO.nEL1809T09State <> 8 THEN
		GVL_Alarms.arrEventFlag[167]:= TRUE;
	ELSIF GVL_Safety.SafetyInputs.bMachineReset THEN
		GVL_Alarms.arrEventFlag[167]:= FALSE;	
END_IF


//*********************************************************END SECTION****************************************************************

//------_________________________-----------------------------------------------------------------------------------------------------
//----- Related to System Faults -----------------------------------------------------------------------------------------------------

(* SF-200: System Powered Off (PLC on Battery) *)
tonSF200Delay( IN := bSF200Alarm, PT := T#3S);

bSF200Alarm := NOT (GVL_IO.gDigInputs.b24VPowerSupplyOK AND GVL_IO.gDigInputs.b24VPowerSupplyOKBck AND GVL_IO.gDigInputs.b48VPowerSupplyOK AND GVL_IO.gDigInputs.b48VPowerSupplyOKBck);

IF tonSF200Delay.Q THEN
		GVL_Alarms.arrEventFlag[200]:= TRUE;
	ELSIF GVL_Safety.SafetyInputs.bMachineReset THEN
		GVL_Alarms.arrEventFlag[200]:= FALSE;	
END_IF

(* SF-202: TwinSAFE Fault (EL6910/EL1918/EL2904) *)
IF 	GVL_IO.stEL6910.nEL6910State <> 8 OR GVL_IO.nEL1918T04State <> 8 OR GVL_IO.nEL1918T05State <> 8 OR 
	GVL_IO.nEL1918T06State <> 8 OR GVL_IO.nEL2904T07State <> 8 OR GVL_IO.nEL2904T08State <> 8 OR GVL_IO.nEL2904T19State <> 8 
	THEN
		GVL_Alarms.arrEventFlag[202]:= TRUE;
	ELSIF GVL_Safety.SafetyInputs.bMachineReset THEN
		GVL_Alarms.arrEventFlag[202]:= FALSE;	
END_IF


(* SF-204: Drive STO Active (M1 - M3 or Valves Motors) *)
IF 	NOT GVL_Safety.iMotorsSTOEnabled THEN
		GVL_Alarms.arrEventFlag[204]:= TRUE;
	ELSIF GVL_Safety.SafetyInputs.bMachineReset THEN
		GVL_Alarms.arrEventFlag[204]:= FALSE;	
END_IF

(* SF-212: Scale Communication Error - TCP Connect *)
IF 	GVL_Alarms.bTCPCLientConnectError THEN
		GVL_Alarms.arrEventFlag[212]:= TRUE;
	ELSIF GVL_Safety.SafetyInputs.bMachineReset THEN
		GVL_Alarms.arrEventFlag[212]:= FALSE;	
END_IF

(* SF-213: Scale Communication Error - TCP Send Message *)
IF 	GVL_Alarms.bTCPCLientSendError THEN
		GVL_Alarms.arrEventFlag[213]:= TRUE;
	ELSIF GVL_Safety.SafetyInputs.bMachineReset THEN
		GVL_Alarms.arrEventFlag[213]:= FALSE;	
END_IF

(* SF-214: Scale Communication Error - TCP Receive Message *)
IF 	GVL_Alarms.bTCPCLientReceiveError THEN
		GVL_Alarms.arrEventFlag[214]:= TRUE;
	ELSIF GVL_Safety.SafetyInputs.bMachineReset THEN
		GVL_Alarms.arrEventFlag[214]:= FALSE;	
END_IF

(* SF-215: Scale Communication Error - TCP Close Communication *)
IF 	GVL_Alarms.bTCPCLientCloseError THEN
		GVL_Alarms.arrEventFlag[215]:= TRUE;
	ELSIF GVL_Safety.SafetyInputs.bMachineReset THEN
		GVL_Alarms.arrEventFlag[215]:= FALSE;	
END_IF

//*********************************************************END SECTION****************************************************************

//------_________________________-----------------------------------------------------------------------------------------------------
//----- Related to Process Fails -----------------------------------------------------------------------------------------------------

(* SF-323: CALIBRATION - Calibration JSON File creation Error *)
IF 	GVL_Alarms.bCalJsonCreationError THEN
		GVL_Alarms.arrEventFlag[323]:= TRUE;
	ELSIF GVL_Safety.SafetyInputs.bMachineReset THEN
		GVL_Alarms.arrEventFlag[323]:= FALSE;	
END_IF

//*********************************************************END SECTION****************************************************************

END_PROGRAM

// ---- POUs/3. HMI/PRG_HMIControl.TcPOU
PROGRAM PRG_HMIControl
VAR
//Motor 1 Animation
rM1MotorPosition     : LREAL;  // Real Motor Actual position
rM1MotorPositionPerc : LREAL;  // Motor Actual Position Scaled 0-100
cM1MinPosition       : LREAL := 0.0; // Minimum expected Value
cM1MaxPosition       : LREAL := -320.0; // Maximum expected Value (Default Value)

//Motor 2 Animation
rM2MotorPosition     : LREAL;  // Real Motor Actual position
rM2MotorPositionPerc : LREAL;  // Motor Actual Position Scaled 0-100
cM2MinPosition       : LREAL := 0.0; // Minimum expected Value
cM2MaxPosition       : LREAL := -170.0; // Maximum expected Value (Default Value)

//Pumps Animation and status
aPumpStatus			: ARRAY[1..10] OF ST_ActuatorStatus;
fbBlinkPumpArrowFWD	: ARRAY[1..10] OF FB_Blink;
fbBlinkPumpArrowBWD	: ARRAY[1..10] OF FB_Blink;

//Headbar Machine Mode transition
fbBlinkMachineModeName 	: FB_Blink;
ePrevMode               : E_MachineMode := E_MachineMode.IMEDIATE_FAULT; 
rTrigChange             : R_TRIG;
bStateChanged           : BOOL;
tpChangePulse           : TP; // gera um pulso de PT quando IN sobe
bBlinkMode              : BOOL;

//Doors Animation
fbBlinkDoor	: ARRAY[1..6] OF FB_Blink;
fbHMIScan	: FB_Blink;

//Icons Animation
bFirstIconSet : BOOL := FALSE;

//EStops Buttons
fbBlinkEStopSide	: FB_Blink;
fbBlinkEStopFront	: FB_Blink;

//Solvent status flags
bSolventIssue : BOOL := FALSE;
ton500ms : TON;
i : INT;

//Timers for releasing interlock signals.
tonInterlockReleaseM1 : ton;
tonInterlockReleaseM2 : ton;
tonInterlockReleaseM3 : ton;

//Jars Animation
curTurns         : LREAL;
deltaTurns       : LREAL;
dMl              : LREAL;
dir              : SINT;       // -1 Fill down, +1 Fill up, 0 stopped
effDeltaMl       : LREAL;
valIdx           : INT;
displayMl        : LREAL;
segPrevEff       : LREAL;
segNowEff        : LREAL;
bRecircActive    : BOOL;
END_VAR

VAR CONSTANT
    cJarsCount              : INT   := 10;
    cJarCapacity_ml         : LREAL := 80.0;
    cDeadVolDefault_ml      : LREAL := 20.0;
    cEpsTurns               : LREAL := 1e-6;
    cRecircLowDeg           : LREAL := 4700.0;
    cRecircHighDeg          : LREAL := 4900.0;
    cRecircDisplayMin_ml    : LREAL := 20.0;   // alvo mínimo visual durante recirculação
END_VAR

VAR RETAIN
    // Integração por bomba (estado interno do jar)
    aPrevTurns       : ARRAY[1..10] OF LREAL;
    aPrevInit        : ARRAY[1..10] OF BOOL;
    aJarMl           : ARRAY[1..10] OF LREAL;

    // Segmentação por direção (fora da recirculação)
    aSegDir          : ARRAY[1..10] OF SINT;     // -1 / 0 / +1
    aSegAbsMl        : ARRAY[1..10] OF LREAL;    // mL acumulados no segmento atual (|mL|)
    aSegAbsMlPrev    : ARRAY[1..10] OF LREAL;

    // Ajustes de unidade e dead volume por bomba
    aUnitsPerTurn    : ARRAY[1..10] OF LREAL := [1(360.0),360.0,360.0,360.0,360.0,360.0,360.0,360.0,360.0,360.0]; // graus->volta
    aDeadVolCfg_ml   : ARRAY[1..10] OF LREAL := [1(cDeadVolDefault_ml),
                                                 cDeadVolDefault_ml, cDeadVolDefault_ml, cDeadVolDefault_ml, cDeadVolDefault_ml,
                                                 cDeadVolDefault_ml, cDeadVolDefault_ml, cDeadVolDefault_ml, cDeadVolDefault_ml, cDeadVolDefault_ml];

    // Exibição durante recirculação
    aRecircWasActive : ARRAY[1..10] OF BOOL;     // para detectar borda de entrada/saída
    aRecircBaseMl    : ARRAY[1..10] OF LREAL;    // patamar antes de entrar em recirculação
    aDispMl          : ARRAY[1..10] OF LREAL;    // nível exibido (pode divergir de aJarMl na recirculação)
END_VAR

//Buttons Indicators -------------------------------------------------------------------------------------------------
GVL_HMI.HMIDigOutputs.bHMIResetButton 	:= GVL_IO.gDigOutputs.bResetIndicator;
GVL_HMI.HMIDigOutputs.bHMIStartButton	:= GVL_IO.gDigOutputs.bStartIndicator;
fbBlinkEStopSide(bEnable := NOT (GVL_Safety.SafetyInputs.bEStopSideCh1 OR GVL_Safety.SafetyInputs.bEStopSideCh2), tPeriod := T#1S); //EStop Button located on side Flashing FB
fbBlinkEStopFront(bEnable := NOT (GVL_Safety.SafetyInputs.bEStopHMICh1 OR GVL_Safety.SafetyInputs.bEStopHMICh2), tPeriod := T#1S);  //EStop Button located on front Flashing FB
GVL_HMI.HMIDigOutputs.bHMIEStopSide		:= fbBlinkEStopSide.bBlink;
GVL_HMI.HMIDigOutputs.bHMIEStopFront	:= fbBlinkEStopFront.bBlink;

(* Alarm Lamp Indicator for HMI --------------------------------------------------------------------------------------- *)
GVL_HMI.HMIDigOutputs.bAlarmLampRed 	:= GVL_IO.gDigOutputs.bTowerRedLight; 	//Red Light
GVL_HMI.HMIDigOutputs.bAlarmLampAmbar 	:= GVL_IO.gDigOutputs.bTowerAmberLight; //Ambar Light
GVL_HMI.HMIDigOutputs.bAlarmLampGreen 	:= GVL_IO.gDigOutputs.bTowerGreenLight; //Green Light

(* <Controls Animation> ------------------------------------------------------------------------------------------------ *)
ACT_M1Animation();
ACT_M2Animation();

(* Head Bar Blinking *) //----------------------------------------------------------------------------------------------------
// 1) State changed?
rTrigChange(CLK := (GVL_HMI.eMachineMode <> ePrevMode));
bStateChanged := rTrigChange.Q;

// 2) Short pulse whe changed
tpChangePulse(IN := bStateChanged, PT := T#500MS);

// 3) Blinking states
bBlinkMode := (GVL_HMI.eMachineMode = E_MachineMode.SYSTEM_READY)
           OR (GVL_HMI.eMachineMode = E_MachineMode.IMEDIATE_FAULT);

// Blinking F
fbBlinkMachineModeName(bEnable := bBlinkMode, tPeriod := T#1S);

// 4) HMI Output
GVL_HMI.bMachineModeBlinking := tpChangePulse.Q OR (bBlinkMode AND fbBlinkMachineModeName.bBlink);

// 5) Update previous machine mode
ePrevMode := GVL_HMI.eMachineMode;

